Yaskawa INFORM job: A_ROOF_UPPER_0614_2_PAINT_51.JBI

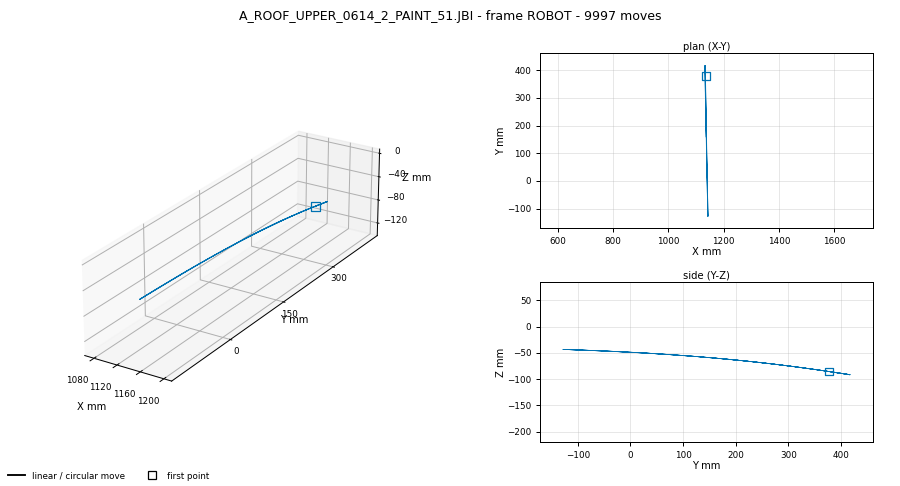
[picture p0: tool path of A_ROOF_UPPER_0614_2_PAINT_51.JBI in frame ROBOT, 9997 of 9997 moves have a stored position in this frame; points joined in program order, loops and branches not executed]
/JOB
//NAME A_ROOF_UPPER_0614_2_PAINT51
//POS
///NPOS 9997,0,0,0,0,0
///TOOL 1
///USER 0
///POSTYPE ROBOT
///RECTAN
///RCONF 1,0,0,0,0,0,0,0,0,0,0,0,0,0,0,0,0,0,0,0,0,0,0,0
C00000=1135.150,378.106,-85.384,-176.923,11.211,149.474
C00001=1135.147,378.354,-85.422,-176.921,11.213,149.474
C00002=1135.142,378.601,-85.459,-176.917,11.216,149.474
C00003=1135.138,378.848,-85.496,-176.915,11.218,149.474
C00004=1135.135,379.096,-85.533,-176.913,11.220,149.474
C00005=1135.131,379.342,-85.571,-176.910,11.222,149.474
C00006=1135.127,379.590,-85.608,-176.907,11.224,149.474
C00007=1135.124,379.837,-85.645,-176.904,11.227,149.474
C00008=1135.120,380.084,-85.682,-176.902,11.229,149.474
C00009=1135.116,380.331,-85.719,-176.899,11.231,149.473
C00010=1135.112,380.578,-85.756,-176.896,11.234,149.473
C00011=1135.108,380.826,-85.794,-176.894,11.236,149.473
C00012=1135.104,381.073,-85.831,-176.891,11.239,149.473
C00013=1135.101,381.320,-85.869,-176.889,11.241,149.473
C00014=1135.097,381.567,-85.906,-176.887,11.243,149.473
C00015=1135.093,381.814,-85.943,-176.883,11.245,149.473
C00016=1135.090,382.062,-85.981,-176.881,11.247,149.473
C00017=1135.086,382.309,-86.017,-176.879,11.249,149.473
C00018=1135.082,382.556,-86.055,-176.876,11.252,149.473
C00019=1135.078,382.803,-86.092,-176.874,11.254,149.473
C00020=1135.075,383.050,-86.130,-176.871,11.256,149.473
C00021=1135.070,383.297,-86.167,-176.869,11.259,149.473
C00022=1135.067,383.545,-86.205,-176.867,11.260,149.473
C00023=1135.063,383.792,-86.241,-176.866,11.262,149.473
C00024=1135.060,384.039,-86.279,-176.865,11.264,149.473
C00025=1135.056,384.286,-86.317,-176.865,11.265,149.473
C00026=1135.052,384.533,-86.354,-176.863,11.266,149.473
C00027=1135.049,384.780,-86.392,-176.862,11.268,149.473
C00028=1135.045,385.027,-86.429,-176.861,11.270,149.474
C00029=1135.042,385.274,-86.467,-176.861,11.271,149.474
C00030=1135.037,385.522,-86.504,-176.860,11.272,149.474
C00031=1135.033,385.769,-86.542,-176.859,11.274,149.474
C00032=1135.030,386.016,-86.580,-176.858,11.276,149.474
C00033=1135.026,386.263,-86.616,-176.857,11.277,149.475
C00034=1135.023,386.510,-86.654,-176.856,11.279,149.475
C00035=1135.018,386.757,-86.691,-176.855,11.280,149.475
C00036=1135.015,387.005,-86.729,-176.854,11.282,149.475
C00037=1135.011,387.252,-86.766,-176.854,11.283,149.476
C00038=1135.007,387.498,-86.804,-176.853,11.285,149.476
C00039=1135.004,387.746,-86.842,-176.853,11.287,149.476
C00040=1134.999,387.993,-86.879,-176.852,11.289,149.476
C00041=1134.996,388.241,-86.917,-176.851,11.290,149.477
C00042=1134.992,388.487,-86.954,-176.851,11.292,149.477
C00043=1134.989,388.700,-86.986,-176.850,11.294,149.477
C00044=1134.986,388.913,-87.019,-176.850,11.295,149.477
C00045=1134.983,389.126,-87.051,-176.849,11.297,149.478
C00046=1134.980,389.339,-87.084,-176.848,11.298,149.478
C00047=1134.976,389.551,-87.116,-176.848,11.300,149.478
C00048=1134.973,389.764,-87.148,-176.847,11.301,149.478
C00049=1134.970,389.977,-87.180,-176.846,11.303,149.479
C00050=1134.967,390.189,-87.213,-176.847,11.305,149.479
C00051=1134.963,390.437,-87.250,-176.846,11.306,149.479
C00052=1134.960,390.684,-87.288,-176.845,11.309,149.480
C00053=1134.956,390.931,-87.326,-176.845,11.310,149.480
C00054=1134.952,391.178,-87.363,-176.845,11.312,149.481
C00055=1134.948,391.426,-87.401,-176.844,11.314,149.481
C00056=1134.945,391.672,-87.439,-176.843,11.316,149.481
C00057=1134.941,391.919,-87.476,-176.844,11.318,149.482
C00058=1134.937,392.167,-87.513,-176.843,11.320,149.482
C00059=1134.933,392.414,-87.552,-176.843,11.322,149.483
C00060=1134.930,392.661,-87.590,-176.842,11.324,149.483
C00061=1134.926,392.908,-87.626,-176.842,11.326,149.483
C00062=1134.922,393.155,-87.664,-176.842,11.328,149.484
C00063=1134.919,393.402,-87.702,-176.841,11.330,149.484
C00064=1134.915,393.650,-87.739,-176.841,11.332,149.485
C00065=1134.911,393.897,-87.777,-176.841,11.334,149.485
C00066=1134.907,394.144,-87.815,-176.841,11.336,149.486
C00067=1134.904,394.391,-87.853,-176.841,11.339,149.486
C00068=1134.900,394.638,-87.890,-176.840,11.341,149.487
C00069=1134.896,394.885,-87.928,-176.840,11.342,149.487
C00070=1134.892,395.133,-87.966,-176.840,11.345,149.488
C00071=1134.889,395.379,-88.004,-176.840,11.347,149.488
C00072=1134.884,395.626,-88.041,-176.840,11.350,149.489
C00073=1134.881,395.874,-88.079,-176.840,11.352,149.490
C00074=1134.878,396.120,-88.116,-176.840,11.354,149.490
C00075=1134.874,396.368,-88.155,-176.840,11.356,149.491
C00076=1134.870,396.614,-88.192,-176.840,11.359,149.491
C00077=1134.866,396.862,-88.229,-176.840,11.361,149.492
C00078=1134.863,397.109,-88.267,-176.839,11.364,149.493
C00079=1134.859,397.356,-88.306,-176.840,11.366,149.493
C00080=1134.855,397.603,-88.343,-176.840,11.368,149.494
C00081=1134.852,397.850,-88.381,-176.840,11.371,149.495
C00082=1134.848,398.097,-88.418,-176.840,11.373,149.495
C00083=1134.844,398.345,-88.456,-176.840,11.376,149.496
C00084=1134.840,398.592,-88.494,-176.840,11.378,149.496
C00085=1134.837,398.839,-88.532,-176.841,11.381,149.497
C00086=1134.833,399.085,-88.570,-176.841,11.383,149.498
C00087=1134.829,399.334,-88.607,-176.841,11.386,149.499
C00088=1134.825,399.580,-88.645,-176.841,11.389,149.499
C00089=1134.822,399.827,-88.683,-176.842,11.391,149.500
C00090=1134.818,400.074,-88.720,-176.842,11.393,149.501
C00091=1134.814,400.322,-88.759,-176.842,11.396,149.502
C00092=1134.810,400.568,-88.797,-176.842,11.399,149.502
C00093=1134.807,400.815,-88.835,-176.843,11.402,149.503
C00094=1134.803,401.063,-88.871,-176.843,11.405,149.504
C00095=1134.799,401.310,-88.910,-176.843,11.407,149.505
C00096=1134.795,401.557,-88.947,-176.844,11.409,149.506
C00097=1134.792,401.804,-88.985,-176.845,11.413,149.507
C00098=1134.788,402.051,-89.023,-176.845,11.416,149.507
C00099=1134.785,402.264,-89.056,-176.845,11.418,149.508
C00100=1134.782,402.476,-89.089,-176.846,11.420,149.509
C00101=1134.779,402.690,-89.121,-176.846,11.423,149.510
C00102=1134.775,402.902,-89.153,-176.846,11.426,149.510
C00103=1134.772,403.114,-89.186,-176.847,11.428,149.511
C00104=1134.769,403.327,-89.219,-176.847,11.431,149.512
C00105=1134.765,403.540,-89.251,-176.848,11.433,149.513
C00106=1134.762,403.753,-89.284,-176.849,11.436,149.514
C00107=1134.759,403.999,-89.322,-176.849,11.439,149.515
C00108=1134.755,404.247,-89.359,-176.850,11.442,149.515
C00109=1134.751,404.494,-89.397,-176.850,11.445,149.516
C00110=1134.747,404.741,-89.435,-176.851,11.448,149.517
C00111=1134.744,404.988,-89.473,-176.852,11.451,149.518
C00112=1134.740,405.235,-89.511,-176.852,11.455,149.519
C00113=1134.736,405.482,-89.549,-176.854,11.457,149.520
C00114=1134.733,405.729,-89.587,-176.854,11.460,149.521
C00115=1134.730,405.977,-89.625,-176.855,11.464,149.522
C00116=1134.725,406.224,-89.663,-176.856,11.467,149.523
C00117=1134.722,406.471,-89.701,-176.857,11.470,149.525
C00118=1134.718,406.717,-89.739,-176.858,11.473,149.526
C00119=1134.715,406.965,-89.777,-176.859,11.477,149.527
C00120=1134.710,407.212,-89.815,-176.859,11.480,149.528
C00121=1134.707,407.459,-89.852,-176.861,11.484,149.529
C00122=1134.703,407.706,-89.889,-176.861,11.487,149.530
C00123=1134.699,407.954,-89.928,-176.862,11.491,149.531
C00124=1134.695,408.200,-89.966,-176.863,11.494,149.532
C00125=1134.692,408.447,-90.004,-176.865,11.498,149.534
C00126=1134.688,408.694,-90.042,-176.866,11.501,149.535
C00127=1134.684,408.942,-90.080,-176.867,11.505,149.536
C00128=1134.681,409.189,-90.118,-176.868,11.508,149.537
C00129=1134.677,409.436,-90.156,-176.869,11.512,149.538
C00130=1134.674,409.683,-90.194,-176.870,11.515,149.540
C00131=1134.670,409.930,-90.231,-176.871,11.519,149.541
C00132=1134.666,410.177,-90.270,-176.873,11.523,149.542
C00133=1134.662,410.424,-90.307,-176.874,11.526,149.543
C00134=1134.659,410.671,-90.345,-176.875,11.530,149.545
C00135=1134.654,410.918,-90.383,-176.876,11.534,149.546
C00136=1134.651,411.165,-90.421,-176.877,11.538,149.547
C00137=1134.648,411.412,-90.459,-176.879,11.542,149.549
C00138=1134.643,411.659,-90.498,-176.880,11.546,149.550
C00139=1134.640,411.907,-90.535,-176.881,11.550,149.551
C00140=1134.636,412.153,-90.573,-176.883,11.554,149.553
C00141=1134.633,412.401,-90.612,-176.884,11.558,149.554
C00142=1134.629,412.647,-90.649,-176.886,11.562,149.556
C00143=1134.626,412.895,-90.687,-176.887,11.566,149.557
C00144=1134.621,413.141,-90.725,-176.889,11.569,149.558
C00145=1134.618,413.389,-90.763,-176.890,11.573,149.560
C00146=1134.615,413.636,-90.801,-176.892,11.578,149.561
C00147=1134.610,413.883,-90.839,-176.893,11.582,149.563
C00148=1134.607,414.130,-90.877,-176.895,11.586,149.564
C00149=1134.603,414.377,-90.915,-176.896,11.590,149.566
C00150=1134.600,414.624,-90.953,-176.898,11.595,149.567
C00151=1134.598,414.871,-90.991,-176.900,11.599,149.569
C00152=1134.597,415.119,-91.029,-176.901,11.604,149.571
C00153=1134.596,415.365,-91.067,-176.903,11.608,149.572
C00154=1134.595,415.613,-91.104,-176.905,11.612,149.574
C00155=1134.595,415.825,-91.136,-176.907,11.616,149.575
C00156=1134.596,416.038,-91.169,-176.908,11.620,149.576
C00157=1134.597,416.250,-91.201,-176.910,11.623,149.578
C00158=1134.599,416.463,-91.233,-176.912,11.627,149.579
C00159=1134.601,416.676,-91.265,-176.913,11.631,149.581
C00160=1134.603,416.888,-91.296,-176.915,11.635,149.582
C00161=1134.606,417.101,-91.328,-176.917,11.639,149.584
C00162=1134.609,417.314,-91.359,-176.919,11.642,149.585
C00163=1134.191,417.313,-91.423,-176.911,11.647,149.584
C00164=1134.187,417.101,-91.391,-176.909,11.643,149.583
C00165=1134.184,416.888,-91.359,-176.907,11.639,149.581
C00166=1134.181,416.675,-91.327,-176.906,11.635,149.580
C00167=1134.179,416.462,-91.295,-176.905,11.631,149.579
C00168=1134.178,416.250,-91.263,-176.903,11.628,149.577
C00169=1134.176,416.037,-91.231,-176.901,11.623,149.576
C00170=1134.176,415.825,-91.199,-176.900,11.620,149.574
C00171=1134.176,415.613,-91.167,-176.898,11.616,149.573
C00172=1134.176,415.365,-91.128,-176.896,11.611,149.571
C00173=1134.177,415.118,-91.091,-176.895,11.607,149.570
C00174=1134.179,414.871,-91.053,-176.893,11.603,149.568
C00175=1134.181,414.624,-91.016,-176.891,11.599,149.567
C00176=1134.184,414.377,-90.978,-176.889,11.595,149.565
C00177=1134.187,414.129,-90.940,-176.889,11.590,149.564
C00178=1134.191,413.883,-90.902,-176.887,11.586,149.562
C00179=1134.194,413.636,-90.864,-176.885,11.582,149.561
C00180=1134.198,413.388,-90.826,-176.883,11.578,149.559
C00181=1134.202,413.141,-90.788,-176.883,11.573,149.558
C00182=1134.206,412.894,-90.749,-176.881,11.569,149.556
C00183=1134.209,412.648,-90.711,-176.880,11.566,149.555
C00184=1134.213,412.401,-90.673,-176.878,11.561,149.554
C00185=1134.217,412.154,-90.635,-176.876,11.557,149.552
C00186=1134.220,411.907,-90.597,-176.875,11.554,149.551
C00187=1134.224,411.659,-90.559,-176.874,11.549,149.550
C00188=1134.228,411.412,-90.521,-176.873,11.545,149.548
C00189=1134.231,411.165,-90.483,-176.871,11.541,149.547
C00190=1134.235,410.919,-90.446,-176.870,11.538,149.546
C00191=1134.239,410.671,-90.407,-176.869,11.534,149.544
C00192=1134.243,410.424,-90.369,-176.868,11.531,149.543
C00193=1134.247,410.177,-90.331,-176.866,11.527,149.542
C00194=1134.250,409.930,-90.293,-176.866,11.522,149.540
C00195=1134.254,409.683,-90.255,-176.865,11.519,149.539
C00196=1134.258,409.435,-90.217,-176.863,11.515,149.538
C00197=1134.261,409.189,-90.179,-176.862,11.511,149.537
C00198=1134.265,408.942,-90.141,-176.861,11.508,149.535
C00199=1134.269,408.695,-90.103,-176.860,11.504,149.534
C00200=1134.272,408.447,-90.065,-176.859,11.501,149.533
C00201=1134.276,408.201,-90.028,-176.858,11.497,149.532
C00202=1134.280,407.953,-89.989,-176.857,11.494,149.531
C00203=1134.283,407.706,-89.951,-176.856,11.490,149.530
C00204=1134.287,407.459,-89.914,-176.855,11.487,149.529
C00205=1134.290,407.212,-89.876,-176.854,11.484,149.527
C00206=1134.295,406.965,-89.838,-176.853,11.480,149.526
C00207=1134.298,406.717,-89.800,-176.852,11.477,149.525
C00208=1134.302,406.471,-89.763,-176.852,11.474,149.524
C00209=1134.306,406.223,-89.724,-176.850,11.470,149.523
C00210=1134.310,405.977,-89.687,-176.850,11.467,149.522
C00211=1134.313,405.729,-89.649,-176.849,11.464,149.521
C00212=1134.317,405.482,-89.610,-176.848,11.460,149.520
C00213=1134.321,405.235,-89.573,-176.848,11.457,149.519
C00214=1134.324,404.988,-89.535,-176.847,11.454,149.518
C00215=1134.328,404.741,-89.496,-176.846,11.451,149.517
C00216=1134.332,404.494,-89.458,-176.846,11.448,149.516
C00217=1134.335,404.247,-89.421,-176.845,11.445,149.515
C00218=1134.338,404.000,-89.383,-176.845,11.441,149.514
C00219=1134.343,403.753,-89.345,-176.844,11.438,149.513
C00220=1134.346,403.540,-89.312,-176.844,11.436,149.512
C00221=1134.350,403.327,-89.280,-176.843,11.434,149.512
C00222=1134.353,403.115,-89.247,-176.843,11.431,149.511
C00223=1134.355,402.902,-89.215,-176.842,11.428,149.510
C00224=1134.359,402.690,-89.182,-176.841,11.426,149.509
C00225=1134.362,402.477,-89.149,-176.841,11.423,149.509
C00226=1134.365,402.264,-89.117,-176.841,11.420,149.508
C00227=1134.368,402.051,-89.084,-176.841,11.419,149.507
C00228=1134.372,401.805,-89.046,-176.840,11.415,149.506
C00229=1134.376,401.556,-89.009,-176.840,11.412,149.505
C00230=1134.380,401.310,-88.971,-176.839,11.410,149.504
C00231=1134.383,401.063,-88.933,-176.839,11.407,149.504
C00232=1134.387,400.816,-88.895,-176.839,11.404,149.503
C00233=1134.391,400.568,-88.857,-176.839,11.401,149.502
C00234=1134.394,400.322,-88.819,-176.838,11.398,149.501
C00235=1134.398,400.075,-88.781,-176.838,11.395,149.500
C00236=1134.401,399.828,-88.744,-176.838,11.393,149.500
C00237=1134.406,399.580,-88.706,-176.837,11.391,149.499
C00238=1134.409,399.333,-88.668,-176.837,11.388,149.498
C00239=1134.413,399.086,-88.630,-176.837,11.385,149.498
C00240=1134.416,398.839,-88.593,-176.837,11.383,149.497
C00241=1134.420,398.592,-88.554,-176.837,11.380,149.496
C00242=1134.424,398.345,-88.517,-176.837,11.378,149.496
C00243=1134.428,398.097,-88.480,-176.837,11.375,149.495
C00244=1134.431,397.851,-88.442,-176.837,11.372,149.494
C00245=1134.435,397.603,-88.403,-176.836,11.370,149.494
C00246=1134.439,397.357,-88.366,-176.836,11.368,149.493
C00247=1134.442,397.109,-88.328,-176.836,11.365,149.492
C00248=1134.446,396.862,-88.291,-176.836,11.363,149.492
C00249=1134.450,396.615,-88.253,-176.837,11.360,149.491
C00250=1134.454,396.368,-88.215,-176.837,11.358,149.490
C00251=1134.457,396.121,-88.177,-176.836,11.356,149.490
C00252=1134.461,395.874,-88.139,-176.837,11.354,149.489
C00253=1134.465,395.626,-88.102,-176.837,11.351,149.489
C00254=1134.469,395.379,-88.064,-176.837,11.349,149.488
C00255=1134.472,395.132,-88.026,-176.837,11.347,149.488
C00256=1134.476,394.886,-87.989,-176.838,11.344,149.487
C00257=1134.480,394.639,-87.951,-176.837,11.343,149.487
C00258=1134.484,394.391,-87.913,-176.838,11.340,149.486
C00259=1134.488,394.144,-87.876,-176.838,11.338,149.485
C00260=1134.491,393.897,-87.838,-176.838,11.336,149.485
C00261=1134.495,393.650,-87.800,-176.839,11.333,149.485
C00262=1134.498,393.402,-87.763,-176.839,11.332,149.484
C00263=1134.503,393.156,-87.725,-176.839,11.330,149.484
C00264=1134.506,392.908,-87.687,-176.840,11.327,149.483
C00265=1134.510,392.662,-87.649,-176.840,11.325,149.483
C00266=1134.513,392.414,-87.612,-176.841,11.323,149.482
C00267=1134.517,392.167,-87.574,-176.840,11.322,149.482
C00268=1134.521,391.920,-87.536,-176.841,11.319,149.481
C00269=1134.525,391.673,-87.499,-176.841,11.317,149.481
C00270=1134.528,391.425,-87.461,-176.842,11.315,149.481
C00271=1134.532,391.179,-87.423,-176.843,11.313,149.480
C00272=1134.536,390.932,-87.386,-176.842,11.312,149.480
C00273=1134.539,390.684,-87.349,-176.843,11.310,149.480
C00274=1134.543,390.438,-87.311,-176.844,11.307,149.479
C00275=1134.547,390.190,-87.273,-176.845,11.306,149.479
C00276=1134.550,389.977,-87.241,-176.845,11.304,149.479
C00277=1134.553,389.764,-87.208,-176.846,11.302,149.478
C00278=1134.557,389.552,-87.176,-176.846,11.301,149.478
C00279=1134.560,389.339,-87.144,-176.846,11.299,149.478
C00280=1134.563,389.126,-87.111,-176.847,11.298,149.477
C00281=1134.566,388.913,-87.080,-176.847,11.296,149.477
C00282=1134.570,388.701,-87.047,-176.848,11.294,149.477
C00283=1134.573,388.488,-87.014,-176.849,11.293,149.477
C00284=1134.577,388.241,-86.977,-176.849,11.291,149.476
C00285=1134.580,387.993,-86.939,-176.850,11.289,149.476
C00286=1134.584,387.747,-86.902,-176.851,11.288,149.476
C00287=1134.587,387.499,-86.865,-176.852,11.287,149.476
C00288=1134.592,387.252,-86.826,-176.853,11.285,149.475
C00289=1134.596,387.005,-86.790,-176.853,11.283,149.475
C00290=1134.599,386.758,-86.752,-176.854,11.281,149.475
C00291=1134.603,386.511,-86.714,-176.855,11.280,149.475
C00292=1134.606,386.263,-86.677,-176.856,11.278,149.475
C00293=1134.610,386.017,-86.639,-176.857,11.276,149.474
C00294=1134.614,385.769,-86.602,-176.858,11.274,149.474
C00295=1134.617,385.522,-86.564,-176.858,11.274,149.474
C00296=1134.621,385.276,-86.527,-176.859,11.272,149.474
C00297=1134.625,385.028,-86.490,-176.860,11.270,149.474
C00298=1134.628,384.781,-86.452,-176.861,11.269,149.474
C00299=1134.633,384.533,-86.414,-176.862,11.267,149.473
C00300=1134.636,384.286,-86.377,-176.863,11.266,149.473
C00301=1134.641,384.039,-86.340,-176.864,11.264,149.473
C00302=1134.644,383.792,-86.302,-176.865,11.262,149.473
C00303=1134.648,383.545,-86.265,-176.866,11.261,149.473
C00304=1134.651,383.297,-86.227,-176.868,11.259,149.473
C00305=1134.655,383.051,-86.189,-176.870,11.256,149.473
C00306=1134.659,382.804,-86.153,-176.873,11.254,149.473
C00307=1134.662,382.556,-86.115,-176.875,11.252,149.473
C00308=1134.666,382.309,-86.078,-176.878,11.250,149.473
C00309=1134.670,382.062,-86.041,-176.881,11.248,149.473
C00310=1134.673,381.815,-86.003,-176.883,11.246,149.473
C00311=1134.678,381.568,-85.966,-176.886,11.243,149.473
C00312=1134.681,381.320,-85.928,-176.888,11.241,149.473
C00313=1134.685,381.073,-85.891,-176.890,11.239,149.473
C00314=1134.689,380.827,-85.854,-176.893,11.236,149.473
C00315=1134.692,380.579,-85.817,-176.895,11.234,149.473
C00316=1134.696,380.331,-85.780,-176.899,11.232,149.474
C00317=1134.700,380.085,-85.742,-176.901,11.230,149.474
C00318=1134.704,379.837,-85.705,-176.903,11.228,149.474
C00319=1134.708,379.590,-85.668,-176.906,11.225,149.474
C00320=1134.711,379.343,-85.630,-176.909,11.223,149.474
C00321=1134.715,379.095,-85.593,-176.912,11.220,149.474
C00322=1134.719,378.848,-85.556,-176.914,11.218,149.474
C00323=1134.723,378.602,-85.519,-176.917,11.216,149.474
C00324=1134.727,378.354,-85.482,-176.920,11.214,149.474
C00325=1134.730,378.107,-85.445,-176.922,11.212,149.474
C00326=1134.733,377.860,-85.408,-176.925,11.209,149.474
C00327=1134.738,377.613,-85.371,-176.927,11.207,149.475
C00328=1134.741,377.365,-85.334,-176.931,11.205,149.475
C00329=1134.745,377.118,-85.297,-176.933,11.203,149.475
C00330=1134.749,376.871,-85.260,-176.936,11.200,149.475
C00331=1134.753,376.624,-85.222,-176.939,11.198,149.475
C00332=1134.755,376.411,-85.191,-176.941,11.197,149.475
C00333=1134.759,376.198,-85.159,-176.944,11.195,149.475
C00334=1134.763,375.985,-85.127,-176.946,11.192,149.475
C00335=1134.766,375.772,-85.096,-176.948,11.191,149.476
C00336=1134.769,375.559,-85.063,-176.951,11.189,149.476
C00337=1134.772,375.347,-85.031,-176.953,11.187,149.476
C00338=1134.776,375.134,-85.000,-176.956,11.185,149.476
C00339=1134.779,374.921,-84.968,-176.958,11.183,149.476
C00340=1134.782,374.673,-84.931,-176.961,11.181,149.476
C00341=1134.786,374.426,-84.894,-176.964,11.178,149.476
C00342=1134.790,374.179,-84.857,-176.967,11.176,149.477
C00343=1134.794,373.932,-84.821,-176.970,11.174,149.477
C00344=1134.798,373.685,-84.784,-176.972,11.172,149.477
C00345=1134.801,373.437,-84.747,-176.976,11.169,149.477
C00346=1134.806,373.190,-84.710,-176.978,11.167,149.477
C00347=1134.809,372.943,-84.674,-176.982,11.165,149.477
C00348=1134.813,372.695,-84.637,-176.985,11.162,149.477
C00349=1134.817,372.448,-84.600,-176.987,11.160,149.478
C00350=1134.821,372.200,-84.563,-176.991,11.158,149.478
C00351=1134.824,371.953,-84.527,-176.993,11.156,149.478
C00352=1134.828,371.706,-84.490,-176.997,11.154,149.478
C00353=1134.832,371.459,-84.453,-176.999,11.151,149.478
C00354=1134.835,371.212,-84.417,-177.002,11.149,149.479
C00355=1134.840,370.965,-84.380,-177.005,11.147,149.479
C00356=1134.843,370.717,-84.343,-177.009,11.144,149.479
C00357=1134.846,370.470,-84.306,-177.011,11.143,149.479
C00358=1134.850,370.223,-84.270,-177.015,11.140,149.480
C00359=1134.855,369.975,-84.233,-177.018,11.138,149.480
C00360=1134.858,369.728,-84.197,-177.021,11.136,149.480
C00361=1134.862,369.481,-84.160,-177.024,11.133,149.480
C00362=1134.866,369.234,-84.123,-177.027,11.131,149.480
C00363=1134.869,368.986,-84.087,-177.030,11.128,149.480
C00364=1134.874,368.739,-84.051,-177.033,11.126,149.481
C00365=1134.877,368.492,-84.014,-177.036,11.124,149.481
C00366=1134.881,368.245,-83.978,-177.039,11.122,149.481
C00367=1134.885,367.997,-83.941,-177.043,11.119,149.481
C00368=1134.889,367.750,-83.905,-177.045,11.117,149.482
C00369=1134.893,367.503,-83.868,-177.049,11.115,149.482
C00370=1134.896,367.256,-83.832,-177.052,11.112,149.482
C00371=1134.901,367.008,-83.796,-177.055,11.110,149.482
C00372=1134.904,366.761,-83.760,-177.058,11.109,149.483
C00373=1134.908,366.514,-83.723,-177.062,11.106,149.483
C00374=1134.912,366.265,-83.686,-177.065,11.104,149.483
C00375=1134.915,366.018,-83.650,-177.068,11.101,149.483
C00376=1134.920,365.771,-83.614,-177.072,11.099,149.483
C00377=1134.923,365.524,-83.578,-177.075,11.096,149.484
C00378=1134.927,365.277,-83.541,-177.078,11.095,149.484
C00379=1134.931,365.029,-83.505,-177.081,11.092,149.484
C00380=1134.934,364.782,-83.469,-177.084,11.090,149.484
C00381=1134.939,364.534,-83.433,-177.088,11.087,149.485
C00382=1134.942,364.288,-83.396,-177.091,11.085,149.485
C00383=1134.946,364.040,-83.360,-177.095,11.083,149.485
C00384=1134.950,363.793,-83.324,-177.098,11.080,149.485
C00385=1134.954,363.545,-83.288,-177.101,11.078,149.486
C00386=1134.957,363.298,-83.252,-177.104,11.075,149.486
C00387=1134.961,363.051,-83.216,-177.107,11.073,149.486
C00388=1134.965,362.838,-83.184,-177.110,11.071,149.486
C00389=1134.968,362.624,-83.154,-177.113,11.069,149.487
C00390=1134.971,362.412,-83.122,-177.116,11.067,149.487
C00391=1134.975,362.198,-83.092,-177.119,11.065,149.487
C00392=1134.978,361.986,-83.061,-177.122,11.063,149.487
C00393=1134.981,361.773,-83.030,-177.125,11.061,149.488
C00394=1134.985,361.560,-82.998,-177.128,11.059,149.488
C00395=1134.988,361.346,-82.968,-177.131,11.057,149.488
C00396=1134.991,361.099,-82.931,-177.134,11.054,149.488
C00397=1134.995,360.852,-82.896,-177.138,11.052,149.488
C00398=1135.000,360.604,-82.860,-177.141,11.049,149.489
C00399=1135.003,360.357,-82.824,-177.145,11.047,149.489
C00400=1135.007,360.110,-82.788,-177.148,11.045,149.489
C00401=1135.010,359.862,-82.752,-177.151,11.042,149.489
C00402=1135.015,359.614,-82.716,-177.155,11.040,149.490
C00403=1135.018,359.367,-82.681,-177.158,11.038,149.490
C00404=1135.022,359.120,-82.644,-177.162,11.035,149.490
C00405=1135.026,358.872,-82.608,-177.165,11.033,149.491
C00406=1135.030,358.625,-82.573,-177.169,11.030,149.491
C00407=1135.034,358.378,-82.537,-177.173,11.027,149.491
C00408=1135.038,358.130,-82.502,-177.176,11.025,149.491
C00409=1135.041,357.883,-82.466,-177.179,11.022,149.492
C00410=1135.045,357.636,-82.429,-177.183,11.020,149.492
C00411=1135.049,357.388,-82.394,-177.186,11.018,149.492
C00412=1135.053,357.141,-82.358,-177.190,11.015,149.492
C00413=1135.056,356.893,-82.323,-177.194,11.012,149.493
C00414=1135.060,356.646,-82.287,-177.197,11.010,149.493
C00415=1135.065,356.399,-82.252,-177.200,11.008,149.493
C00416=1135.069,356.151,-82.216,-177.204,11.005,149.494
C00417=1135.072,355.904,-82.180,-177.208,11.002,149.494
C00418=1135.076,355.656,-82.145,-177.211,11.000,149.494
C00419=1135.080,355.409,-82.109,-177.215,10.998,149.494
C00420=1135.083,355.161,-82.074,-177.218,10.995,149.495
C00421=1135.088,354.914,-82.039,-177.222,10.992,149.495
C00422=1135.091,354.667,-82.003,-177.226,10.989,149.495
C00423=1135.095,354.419,-81.968,-177.229,10.987,149.495
C00424=1135.100,354.171,-81.932,-177.233,10.984,149.496
C00425=1135.104,353.924,-81.897,-177.237,10.982,149.496
C00426=1135.108,353.677,-81.861,-177.240,10.979,149.496
C00427=1135.111,353.429,-81.826,-177.244,10.976,149.497
C00428=1135.115,353.182,-81.790,-177.248,10.974,149.497
C00429=1135.119,352.934,-81.755,-177.251,10.972,149.497
C00430=1135.123,352.687,-81.720,-177.255,10.968,149.497
C00431=1135.127,352.439,-81.685,-177.258,10.966,149.498
C00432=1135.130,352.192,-81.649,-177.263,10.963,149.498
C00433=1135.134,351.944,-81.614,-177.266,10.961,149.498
C00434=1135.139,351.697,-81.579,-177.269,10.958,149.498
C00435=1135.142,351.449,-81.544,-177.274,10.955,149.499
C00436=1135.146,351.202,-81.508,-177.277,10.953,149.499
C00437=1135.151,350.954,-81.474,-177.281,10.949,149.499
C00438=1135.154,350.707,-81.438,-177.285,10.947,149.500
C00439=1135.158,350.459,-81.402,-177.289,10.944,149.500
C00440=1135.162,350.212,-81.369,-177.292,10.942,149.500
C00441=1135.165,349.965,-81.333,-177.296,10.939,149.500
C00442=1135.169,349.717,-81.297,-177.300,10.936,149.501
C00443=1135.174,349.470,-81.263,-177.304,10.933,149.501
C00444=1135.177,349.257,-81.232,-177.306,10.931,149.501
C00445=1135.180,349.043,-81.202,-177.310,10.929,149.501
C00446=1135.184,348.829,-81.172,-177.312,10.927,149.501
C00447=1135.187,348.616,-81.142,-177.315,10.924,149.502
C00448=1135.191,348.404,-81.112,-177.317,10.922,149.502
C00449=1135.194,348.191,-81.081,-177.320,10.921,149.502
C00450=1135.197,347.977,-81.052,-177.323,10.918,149.502
C00451=1135.200,347.764,-81.022,-177.326,10.916,149.502
C00452=1135.204,347.517,-80.986,-177.329,10.914,149.502
C00453=1135.208,347.269,-80.952,-177.332,10.911,149.503
C00454=1135.212,347.021,-80.917,-177.336,10.909,149.503
C00455=1135.216,346.774,-80.882,-177.339,10.906,149.503
C00456=1135.220,346.526,-80.847,-177.342,10.904,149.503
C00457=1135.224,346.279,-80.812,-177.346,10.902,149.504
C00458=1135.228,346.031,-80.777,-177.349,10.899,149.504
C00459=1135.232,345.783,-80.742,-177.352,10.896,149.504
C00460=1135.236,345.536,-80.708,-177.355,10.894,149.504
C00461=1135.240,345.288,-80.673,-177.359,10.891,149.504
C00462=1135.244,345.041,-80.639,-177.362,10.889,149.505
C00463=1135.248,344.793,-80.603,-177.365,10.886,149.505
C00464=1135.252,344.546,-80.569,-177.368,10.884,149.505
C00465=1135.256,344.298,-80.534,-177.372,10.882,149.505
C00466=1135.260,344.050,-80.499,-177.375,10.879,149.505
C00467=1135.263,343.804,-80.465,-177.378,10.876,149.506
C00468=1135.267,343.555,-80.430,-177.381,10.874,149.506
C00469=1135.272,343.308,-80.396,-177.385,10.871,149.506
C00470=1135.275,343.060,-80.361,-177.388,10.869,149.506
C00471=1135.279,342.813,-80.327,-177.391,10.866,149.507
C00472=1135.283,342.565,-80.291,-177.395,10.864,149.507
C00473=1135.287,342.318,-80.257,-177.397,10.861,149.507
C00474=1135.291,342.070,-80.223,-177.401,10.859,149.507
C00475=1135.296,341.823,-80.188,-177.404,10.856,149.507
C00476=1135.299,341.575,-80.154,-177.407,10.854,149.508
C00477=1135.303,341.327,-80.119,-177.411,10.851,149.508
C00478=1135.307,341.079,-80.085,-177.414,10.849,149.508
C00479=1135.311,340.832,-80.051,-177.417,10.846,149.508
C00480=1135.316,340.585,-80.016,-177.420,10.844,149.508
C00481=1135.319,340.337,-79.982,-177.424,10.841,149.508
C00482=1135.323,340.090,-79.948,-177.427,10.839,149.509
C00483=1135.327,339.842,-79.913,-177.430,10.836,149.509
C00484=1135.331,339.594,-79.879,-177.434,10.834,149.509
C00485=1135.335,339.346,-79.844,-177.436,10.831,149.509
C00486=1135.339,339.099,-79.810,-177.440,10.829,149.509
C00487=1135.343,338.851,-79.775,-177.443,10.826,149.510
C00488=1135.347,338.604,-79.741,-177.446,10.824,149.510
C00489=1135.351,338.356,-79.707,-177.450,10.821,149.510
C00490=1135.355,338.109,-79.673,-177.453,10.819,149.510
C00491=1135.359,337.861,-79.638,-177.456,10.816,149.510
C00492=1135.362,337.613,-79.604,-177.459,10.814,149.511
C00493=1135.367,337.366,-79.570,-177.463,10.811,149.511
C00494=1135.371,337.119,-79.536,-177.466,10.809,149.511
C00495=1135.374,336.870,-79.502,-177.469,10.806,149.511
C00496=1135.379,336.623,-79.468,-177.472,10.803,149.512
C00497=1135.382,336.375,-79.433,-177.476,10.801,149.512
C00498=1135.387,336.128,-79.399,-177.479,10.799,149.512
C00499=1135.391,335.881,-79.365,-177.482,10.797,149.512
C00500=1135.394,335.667,-79.336,-177.484,10.794,149.512
C00501=1135.397,335.453,-79.306,-177.487,10.792,149.513
C00502=1135.401,335.240,-79.277,-177.490,10.790,149.513
C00503=1135.404,335.027,-79.248,-177.493,10.788,149.513
C00504=1135.408,334.814,-79.218,-177.496,10.785,149.513
C00505=1135.411,334.600,-79.189,-177.498,10.784,149.513
C00506=1135.414,334.387,-79.160,-177.501,10.782,149.513
C00507=1135.418,334.173,-79.130,-177.504,10.779,149.514
C00508=1135.422,333.925,-79.097,-177.507,10.777,149.514
C00509=1135.425,333.678,-79.063,-177.510,10.774,149.514
C00510=1135.430,333.430,-79.029,-177.514,10.771,149.514
C00511=1135.434,333.182,-78.995,-177.517,10.769,149.514
C00512=1135.438,332.935,-78.962,-177.520,10.767,149.515
C00513=1135.441,332.688,-78.927,-177.523,10.764,149.515
C00514=1135.446,332.439,-78.894,-177.526,10.761,149.515
C00515=1135.450,332.192,-78.860,-177.530,10.759,149.515
C00516=1135.453,331.944,-78.826,-177.533,10.756,149.515
C00517=1135.458,331.697,-78.792,-177.536,10.754,149.515
C00518=1135.462,331.449,-78.759,-177.539,10.751,149.516
C00519=1135.466,331.202,-78.725,-177.543,10.749,149.516
C00520=1135.469,330.953,-78.691,-177.546,10.746,149.516
C00521=1135.473,330.706,-78.657,-177.549,10.743,149.516
C00522=1135.478,330.458,-78.624,-177.552,10.741,149.516
C00523=1135.482,330.211,-78.590,-177.555,10.739,149.517
C00524=1135.486,329.963,-78.556,-177.558,10.737,149.517
C00525=1135.490,329.715,-78.523,-177.561,10.734,149.517
C00526=1135.494,329.468,-78.489,-177.564,10.732,149.517
C00527=1135.498,329.220,-78.455,-177.568,10.729,149.518
C00528=1135.502,328.972,-78.421,-177.571,10.726,149.518
C00529=1135.506,328.724,-78.388,-177.574,10.724,149.518
C00530=1135.510,328.476,-78.355,-177.577,10.722,149.518
C00531=1135.514,328.229,-78.321,-177.581,10.719,149.518
C00532=1135.518,327.982,-78.288,-177.584,10.716,149.518
C00533=1135.521,327.733,-78.254,-177.587,10.714,149.519
C00534=1135.526,327.486,-78.220,-177.590,10.711,149.519
C00535=1135.530,327.238,-78.187,-177.593,10.709,149.519
C00536=1135.534,326.990,-78.154,-177.596,10.706,149.519
C00537=1135.538,326.743,-78.120,-177.600,10.704,149.519
C00538=1135.542,326.495,-78.086,-177.603,10.701,149.520
C00539=1135.546,326.247,-78.053,-177.606,10.699,149.520
C00540=1135.550,325.999,-78.020,-177.609,10.696,149.520
C00541=1135.554,325.752,-77.987,-177.613,10.694,149.520
C00542=1135.558,325.504,-77.953,-177.616,10.691,149.520
C00543=1135.562,325.256,-77.920,-177.619,10.688,149.521
C00544=1135.566,325.009,-77.886,-177.622,10.686,149.521
C00545=1135.570,324.761,-77.853,-177.625,10.683,149.521
C00546=1135.574,324.513,-77.820,-177.629,10.681,149.521
C00547=1135.578,324.265,-77.787,-177.632,10.678,149.521
C00548=1135.582,324.017,-77.753,-177.635,10.676,149.522
C00549=1135.586,323.770,-77.720,-177.638,10.673,149.522
C00550=1135.590,323.522,-77.687,-177.641,10.671,149.522
C00551=1135.595,323.274,-77.654,-177.645,10.668,149.522
C00552=1135.599,323.026,-77.621,-177.648,10.665,149.522
C00553=1135.603,322.779,-77.588,-177.651,10.663,149.523
C00554=1135.606,322.531,-77.555,-177.654,10.661,149.523
C00555=1135.610,322.283,-77.522,-177.657,10.658,149.523
C00556=1135.613,322.070,-77.493,-177.660,10.656,149.523
C00557=1135.617,321.856,-77.465,-177.662,10.654,149.523
C00558=1135.620,321.642,-77.436,-177.666,10.652,149.523
C00559=1135.624,321.429,-77.407,-177.668,10.650,149.524
C00560=1135.628,321.216,-77.379,-177.671,10.647,149.524
C00561=1135.631,321.002,-77.350,-177.673,10.645,149.524
C00562=1135.634,320.789,-77.322,-177.676,10.643,149.524
C00563=1135.638,320.575,-77.293,-177.679,10.641,149.524
C00564=1135.642,320.328,-77.260,-177.682,10.638,149.524
C00565=1135.646,320.080,-77.228,-177.685,10.636,149.525
C00566=1135.650,319.832,-77.195,-177.689,10.633,149.525
C00567=1135.654,319.584,-77.162,-177.692,10.630,149.525
C00568=1135.659,319.336,-77.129,-177.695,10.628,149.525
C00569=1135.663,319.089,-77.096,-177.698,10.626,149.525
C00570=1135.666,318.841,-77.063,-177.701,10.623,149.525
C00571=1135.670,318.593,-77.031,-177.704,10.620,149.526
C00572=1135.675,318.345,-76.998,-177.708,10.618,149.526
C00573=1135.679,318.097,-76.964,-177.710,10.616,149.526
C00574=1135.682,317.850,-76.932,-177.713,10.613,149.526
C00575=1135.687,317.602,-76.899,-177.717,10.611,149.527
C00576=1135.691,317.354,-76.866,-177.720,10.608,149.527
C00577=1135.695,317.106,-76.833,-177.723,10.606,149.527
C00578=1135.699,316.858,-76.801,-177.726,10.603,149.527
C00579=1135.703,316.610,-76.768,-177.729,10.601,149.527
C00580=1135.707,316.363,-76.735,-177.733,10.598,149.527
C00581=1135.711,316.115,-76.703,-177.736,10.595,149.528
C00582=1135.715,315.867,-76.670,-177.739,10.593,149.528
C00583=1135.719,315.619,-76.637,-177.742,10.591,149.528
C00584=1135.723,315.371,-76.605,-177.745,10.588,149.528
C00585=1135.727,315.123,-76.572,-177.748,10.585,149.528
C00586=1135.731,314.875,-76.539,-177.752,10.583,149.529
C00587=1135.735,314.628,-76.507,-177.755,10.580,149.529
C00588=1135.740,314.380,-76.475,-177.758,10.578,149.529
C00589=1135.743,314.133,-76.442,-177.761,10.575,149.529
C00590=1135.747,313.884,-76.410,-177.764,10.572,149.529
C00591=1135.752,313.636,-76.377,-177.768,10.570,149.530
C00592=1135.755,313.388,-76.345,-177.771,10.567,149.530
C00593=1135.759,313.141,-76.312,-177.774,10.565,149.530
C00594=1135.763,312.893,-76.280,-177.777,10.562,149.530
C00595=1135.767,312.645,-76.247,-177.780,10.560,149.530
C00596=1135.772,312.397,-76.215,-177.783,10.558,149.531
C00597=1135.776,312.149,-76.183,-177.786,10.555,149.531
C00598=1135.780,311.902,-76.150,-177.789,10.553,149.531
C00599=1135.784,311.653,-76.118,-177.792,10.550,149.531
C00600=1135.788,311.406,-76.085,-177.795,10.548,149.531
C00601=1135.792,311.158,-76.053,-177.799,10.545,149.531
C00602=1135.797,310.910,-76.021,-177.802,10.542,149.532
C00603=1135.800,310.663,-75.988,-177.805,10.540,149.532
C00604=1135.805,310.414,-75.956,-177.808,10.537,149.532
C00605=1135.808,310.166,-75.924,-177.811,10.535,149.532
C00606=1135.813,309.918,-75.891,-177.815,10.532,149.532
C00607=1135.816,309.670,-75.859,-177.817,10.529,149.532
C00608=1135.821,309.423,-75.827,-177.821,10.527,149.533
C00609=1135.825,309.175,-75.795,-177.824,10.524,149.533
C00610=1135.829,308.927,-75.763,-177.827,10.522,149.533
C00611=1135.833,308.679,-75.730,-177.830,10.519,149.533
C00612=1135.837,308.454,-75.701,-177.833,10.517,149.533
C00613=1135.840,308.229,-75.672,-177.836,10.515,149.534
C00614=1135.844,308.004,-75.643,-177.839,10.512,149.534
C00615=1135.847,307.779,-75.614,-177.841,10.510,149.534
C00616=1135.852,307.555,-75.585,-177.845,10.508,149.534
C00617=1135.856,307.329,-75.555,-177.847,10.506,149.534
C00618=1135.860,307.104,-75.527,-177.850,10.503,149.534
C00619=1135.863,306.879,-75.497,-177.853,10.501,149.535
C00620=1135.867,306.631,-75.465,-177.855,10.499,149.535
C00621=1135.871,306.384,-75.434,-177.859,10.496,149.535
C00622=1135.875,306.136,-75.401,-177.862,10.494,149.535
C00623=1135.879,305.888,-75.369,-177.865,10.491,149.535
C00624=1135.883,305.640,-75.338,-177.868,10.489,149.536
C00625=1135.888,305.392,-75.306,-177.871,10.486,149.536
C00626=1135.892,305.144,-75.274,-177.875,10.483,149.536
C00627=1135.895,304.896,-75.242,-177.878,10.481,149.536
C00628=1135.900,304.648,-75.210,-177.881,10.478,149.536
C00629=1135.904,304.400,-75.178,-177.884,10.475,149.536
C00630=1135.908,304.152,-75.146,-177.887,10.473,149.537
C00631=1135.912,303.905,-75.115,-177.891,10.471,149.537
C00632=1135.917,303.657,-75.082,-177.893,10.468,149.537
C00633=1135.920,303.409,-75.050,-177.897,10.465,149.537
C00634=1135.925,303.161,-75.019,-177.900,10.463,149.537
C00635=1135.929,302.913,-74.988,-177.903,10.460,149.538
C00636=1135.933,302.664,-74.955,-177.905,10.458,149.538
C00637=1135.937,302.417,-74.924,-177.909,10.456,149.538
C00638=1135.941,302.169,-74.892,-177.912,10.453,149.538
C00639=1135.945,301.921,-74.860,-177.915,10.451,149.538
C00640=1135.949,301.673,-74.829,-177.918,10.448,149.538
C00641=1135.954,301.424,-74.797,-177.921,10.445,149.539
C00642=1135.958,301.177,-74.765,-177.924,10.443,149.539
C00643=1135.962,300.929,-74.734,-177.927,10.440,149.539
C00644=1135.966,300.682,-74.702,-177.931,10.438,149.539
C00645=1135.970,300.433,-74.671,-177.934,10.435,149.539
C00646=1135.974,300.185,-74.639,-177.937,10.432,149.540
C00647=1135.978,299.938,-74.608,-177.940,10.430,149.540
C00648=1135.983,299.689,-74.576,-177.943,10.427,149.540
C00649=1135.987,299.441,-74.544,-177.946,10.425,149.540
C00650=1135.991,299.193,-74.513,-177.950,10.422,149.540
C00651=1135.996,298.945,-74.482,-177.953,10.419,149.540
C00652=1135.999,298.697,-74.450,-177.955,10.418,149.541
C00653=1136.003,298.449,-74.418,-177.958,10.415,149.541
C00654=1136.008,298.201,-74.387,-177.962,10.412,149.541
C00655=1136.011,297.953,-74.356,-177.964,10.410,149.541
C00656=1136.016,297.705,-74.325,-177.968,10.407,149.541
C00657=1136.020,297.457,-74.293,-177.971,10.405,149.541
C00658=1136.024,297.209,-74.262,-177.974,10.402,149.542
C00659=1136.028,296.961,-74.230,-177.977,10.399,149.542
C00660=1136.032,296.714,-74.199,-177.980,10.397,149.542
C00661=1136.036,296.465,-74.168,-177.983,10.394,149.542
C00662=1136.041,296.218,-74.136,-177.987,10.392,149.542
C00663=1136.045,295.969,-74.105,-177.990,10.389,149.543
C00664=1136.066,294.691,-73.943,-177.108,8.658,148.873
C00665=1136.070,294.443,-73.913,-177.111,8.654,148.872
C00666=1136.074,294.195,-73.882,-177.114,8.650,148.872
C00667=1136.079,293.947,-73.851,-177.116,8.648,148.872
C00668=1136.082,293.699,-73.821,-177.119,8.643,148.872
C00669=1136.087,293.451,-73.790,-177.122,8.641,148.872
C00670=1136.091,293.203,-73.759,-177.124,8.637,148.872
C00671=1136.095,292.954,-73.729,-177.127,8.633,148.872
C00672=1136.099,292.706,-73.698,-177.130,8.630,148.872
C00673=1136.104,292.458,-73.667,-177.133,8.626,148.872
C00674=1136.107,292.210,-73.637,-177.135,8.623,148.871
C00675=1136.112,291.962,-73.606,-177.138,8.620,148.872
C00676=1136.116,291.714,-73.575,-177.141,8.616,148.871
C00677=1136.120,291.466,-73.545,-177.144,8.613,148.871
C00678=1136.124,291.218,-73.514,-177.146,8.610,148.871
C00679=1136.129,290.969,-73.484,-177.149,8.606,148.871
C00680=1136.133,290.722,-73.454,-177.152,8.603,148.871
C00681=1136.137,290.473,-73.422,-177.154,8.600,148.871
C00682=1136.141,290.225,-73.392,-177.157,8.596,148.871
C00683=1136.146,289.977,-73.361,-177.160,8.593,148.871
C00684=1136.149,289.730,-73.331,-177.162,8.589,148.871
C00685=1136.154,289.480,-73.301,-177.166,8.586,148.871
C00686=1136.158,289.233,-73.271,-177.168,8.582,148.870
C00687=1136.162,288.985,-73.240,-177.171,8.579,148.870
C00688=1136.167,288.737,-73.209,-177.174,8.575,148.870
C00689=1136.171,288.489,-73.179,-177.176,8.572,148.870
C00690=1136.175,288.240,-73.149,-177.179,8.569,148.870
C00691=1136.179,287.992,-73.118,-177.182,8.565,148.870
C00692=1136.184,287.744,-73.088,-177.185,8.562,148.870
C00693=1136.188,287.468,-73.055,-177.188,8.558,148.870
C00694=1136.193,287.193,-73.021,-177.191,8.554,148.870
C00695=1136.197,286.918,-72.987,-177.193,8.551,148.870
C00696=1136.202,286.641,-72.954,-177.197,8.547,148.870
C00697=1136.206,286.394,-72.923,-177.200,8.543,148.869
C00698=1136.210,286.146,-72.893,-177.202,8.540,148.869
C00699=1136.215,285.897,-72.863,-177.205,8.537,148.869
C00700=1136.218,285.649,-72.833,-177.208,8.533,148.869
C00701=1136.223,285.400,-72.803,-177.211,8.530,148.869
C00702=1136.227,285.153,-72.772,-177.213,8.527,148.869
C00703=1136.231,284.904,-72.743,-177.216,8.524,148.869
C00704=1136.236,284.657,-72.712,-177.219,8.520,148.869
C00705=1136.240,284.408,-72.683,-177.221,8.517,148.869
C00706=1136.245,284.160,-72.652,-177.224,8.514,148.869
C00707=1136.249,283.912,-72.623,-177.227,8.510,148.869
C00708=1136.253,283.664,-72.592,-177.229,8.507,148.869
C00709=1136.257,283.415,-72.562,-177.232,8.504,148.869
C00710=1136.261,283.167,-72.532,-177.235,8.500,148.868
C00711=1136.265,282.919,-72.502,-177.238,8.497,148.868
C00712=1136.270,282.671,-72.472,-177.240,8.494,148.868
C00713=1136.274,282.423,-72.442,-177.243,8.491,148.868
C00714=1136.278,282.175,-72.413,-177.246,8.487,148.868
C00715=1136.282,281.927,-72.382,-177.249,8.484,148.868
C00716=1136.287,281.678,-72.352,-177.252,8.481,148.868
C00717=1136.291,281.430,-72.323,-177.255,8.477,148.868
C00718=1136.295,281.183,-72.293,-177.257,8.474,148.868
C00719=1136.299,280.934,-72.263,-177.260,8.471,148.868
C00720=1136.304,280.686,-72.233,-177.262,8.468,148.868
C00721=1136.308,280.438,-72.203,-177.265,8.464,148.868
C00722=1136.312,280.190,-72.174,-177.268,8.461,148.868
C00723=1136.316,279.942,-72.144,-177.271,8.457,148.868
C00724=1136.321,279.693,-72.114,-177.274,8.454,148.868
C00725=1136.325,279.445,-72.084,-177.276,8.450,148.868
C00726=1136.329,279.197,-72.055,-177.279,8.447,148.868
C00727=1136.333,278.949,-72.025,-177.282,8.445,148.868
C00728=1136.338,278.701,-71.996,-177.285,8.440,148.867
C00729=1136.342,278.452,-71.966,-177.288,8.438,148.868
C00730=1136.346,278.204,-71.937,-177.290,8.434,148.867
C00731=1136.351,277.956,-71.906,-177.293,8.431,148.867
C00732=1136.355,277.708,-71.877,-177.296,8.427,148.867
C00733=1136.359,277.459,-71.847,-177.298,8.424,148.867
C00734=1136.363,277.211,-71.818,-177.301,8.421,148.867
C00735=1136.367,276.963,-71.788,-177.304,8.418,148.867
C00736=1136.372,276.715,-71.759,-177.307,8.414,148.867
C00737=1136.376,276.466,-71.729,-177.309,8.411,148.867
C00738=1136.380,276.218,-71.700,-177.312,8.408,148.867
C00739=1136.384,275.970,-71.670,-177.314,8.405,148.867
C00740=1136.388,275.722,-71.641,-177.318,8.401,148.867
C00741=1136.392,275.473,-71.611,-177.321,8.398,148.867
C00742=1136.397,275.225,-71.582,-177.323,8.395,148.867
C00743=1136.401,274.977,-71.553,-177.326,8.392,148.867
C00744=1136.406,274.729,-71.523,-177.329,8.388,148.867
C00745=1136.410,274.481,-71.494,-177.332,8.385,148.867
C00746=1136.414,274.233,-71.465,-177.334,8.382,148.867
C00747=1136.418,273.984,-71.435,-177.337,8.379,148.867
C00748=1136.422,273.736,-71.406,-177.339,8.376,148.867
C00749=1136.427,273.488,-71.376,-177.343,8.372,148.867
C00750=1136.431,273.240,-71.347,-177.345,8.369,148.867
C00751=1136.435,272.991,-71.318,-177.348,8.366,148.867
C00752=1136.439,272.742,-71.289,-177.351,8.363,148.867
C00753=1136.444,272.495,-71.259,-177.354,8.359,148.866
C00754=1136.448,272.247,-71.230,-177.356,8.356,148.867
C00755=1136.452,271.998,-71.201,-177.359,8.353,148.866
C00756=1136.457,271.749,-71.172,-177.362,8.350,148.866
C00757=1136.461,271.501,-71.142,-177.364,8.347,148.867
C00758=1136.465,271.253,-71.113,-177.367,8.343,148.866
C00759=1136.469,271.006,-71.084,-177.370,8.340,148.866
C00760=1136.474,270.757,-71.056,-177.373,8.337,148.866
C00761=1136.478,270.509,-71.026,-177.375,8.334,148.866
C00762=1136.482,270.260,-70.997,-177.379,8.330,148.866
C00763=1136.486,270.012,-70.967,-177.381,8.327,148.866
C00764=1136.492,269.764,-70.939,-177.384,8.324,148.866
C00765=1136.495,269.516,-70.910,-177.387,8.321,148.866
C00766=1136.499,269.268,-70.881,-177.389,8.318,148.866
C00767=1136.504,269.019,-70.852,-177.392,8.314,148.866
C00768=1136.508,268.771,-70.823,-177.395,8.311,148.866
C00769=1136.513,268.522,-70.794,-177.398,8.308,148.866
C00770=1136.516,268.274,-70.765,-177.400,8.305,148.866
C00771=1136.521,268.025,-70.736,-177.403,8.302,148.866
C00772=1136.526,267.778,-70.707,-177.406,8.299,148.866
C00773=1136.530,267.530,-70.678,-177.409,8.296,148.866
C00774=1136.534,267.281,-70.650,-177.412,8.292,148.866
C00775=1136.538,267.033,-70.620,-177.414,8.289,148.866
C00776=1136.543,266.785,-70.592,-177.417,8.287,148.866
C00777=1136.547,266.536,-70.562,-177.420,8.283,148.866
C00778=1136.551,266.288,-70.534,-177.423,8.280,148.866
C00779=1136.555,266.039,-70.505,-177.426,8.277,148.866
C00780=1136.560,265.791,-70.477,-177.428,8.273,148.866
C00781=1136.564,265.543,-70.448,-177.431,8.270,148.866
C00782=1136.568,265.294,-70.419,-177.434,8.268,148.866
C00783=1136.573,265.046,-70.391,-177.436,8.265,148.866
C00784=1136.576,264.798,-70.362,-177.439,8.261,148.866
C00785=1136.581,264.549,-70.333,-177.442,8.258,148.866
C00786=1136.586,264.301,-70.305,-177.445,8.255,148.866
C00787=1136.589,264.053,-70.276,-177.448,8.252,148.866
C00788=1136.594,263.804,-70.247,-177.450,8.249,148.866
C00789=1136.599,263.556,-70.219,-177.453,8.246,148.866
C00790=1136.603,263.308,-70.190,-177.456,8.242,148.866
C00791=1136.608,263.060,-70.161,-177.459,8.239,148.866
C00792=1136.611,262.811,-70.133,-177.461,8.236,148.866
C00793=1136.616,262.563,-70.105,-177.464,8.233,148.866
C00794=1136.620,262.315,-70.076,-177.467,8.230,148.866
C00795=1136.624,262.066,-70.047,-177.470,8.227,148.866
C00796=1136.629,261.818,-70.019,-177.473,8.223,148.866
C00797=1136.634,261.544,-69.988,-177.476,8.220,148.866
C00798=1136.639,261.271,-69.956,-177.479,8.216,148.866
C00799=1136.643,260.997,-69.925,-177.482,8.213,148.866
C00800=1136.648,260.723,-69.894,-177.485,8.210,148.866
C00801=1136.652,260.475,-69.865,-177.487,8.206,148.866
C00802=1136.657,260.227,-69.837,-177.490,8.203,148.866
C00803=1136.660,259.979,-69.808,-177.493,8.201,148.866
C00804=1136.665,259.731,-69.780,-177.496,8.198,148.866
C00805=1136.669,259.482,-69.752,-177.499,8.194,148.866
C00806=1136.674,259.233,-69.723,-177.502,8.191,148.866
C00807=1136.678,258.985,-69.695,-177.504,8.188,148.866
C00808=1136.682,258.737,-69.667,-177.507,8.185,148.866
C00809=1136.687,258.488,-69.639,-177.510,8.182,148.866
C00810=1136.691,258.240,-69.610,-177.513,8.179,148.866
C00811=1136.696,257.992,-69.582,-177.515,8.176,148.866
C00812=1136.699,257.743,-69.554,-177.518,8.173,148.866
C00813=1136.704,257.495,-69.526,-177.521,8.169,148.866
C00814=1136.708,257.246,-69.497,-177.524,8.166,148.866
C00815=1136.713,256.998,-69.470,-177.527,8.163,148.867
C00816=1136.716,256.750,-69.442,-177.529,8.160,148.866
C00817=1136.722,256.502,-69.413,-177.532,8.157,148.866
C00818=1136.725,256.253,-69.385,-177.535,8.154,148.867
C00819=1136.730,256.005,-69.357,-177.538,8.151,148.867
C00820=1136.734,255.756,-69.329,-177.540,8.148,148.867
C00821=1136.739,255.508,-69.301,-177.543,8.145,148.867
C00822=1136.743,255.259,-69.273,-177.546,8.141,148.867
C00823=1136.748,255.011,-69.245,-177.549,8.138,148.867
C00824=1136.751,254.763,-69.217,-177.552,8.136,148.867
C00825=1136.756,254.515,-69.189,-177.555,8.133,148.867
C00826=1136.761,254.266,-69.161,-177.557,8.130,148.867
C00827=1136.765,254.017,-69.133,-177.560,8.127,148.867
C00828=1136.769,253.769,-69.105,-177.563,8.124,148.867
C00829=1136.773,253.521,-69.077,-177.565,8.121,148.867
C00830=1136.778,253.272,-69.050,-177.568,8.118,148.867
C00831=1136.782,253.023,-69.022,-177.571,8.115,148.867
C00832=1136.786,252.776,-68.994,-177.574,8.111,148.867
C00833=1136.791,252.528,-68.966,-177.577,8.108,148.867
C00834=1136.795,252.278,-68.939,-177.579,8.105,148.867
C00835=1136.800,252.030,-68.910,-177.582,8.102,148.867
C00836=1136.804,251.782,-68.882,-177.585,8.099,148.867
C00837=1136.808,251.533,-68.855,-177.588,8.096,148.867
C00838=1136.813,251.285,-68.827,-177.591,8.093,148.867
C00839=1136.817,251.036,-68.800,-177.593,8.090,148.867
C00840=1136.821,250.788,-68.772,-177.596,8.087,148.867
C00841=1136.825,250.540,-68.744,-177.599,8.085,148.867
C00842=1136.830,250.291,-68.716,-177.601,8.081,148.867
C00843=1136.835,250.043,-68.688,-177.604,8.078,148.867
C00844=1136.839,249.795,-68.661,-177.607,8.075,148.867
C00845=1136.843,249.546,-68.633,-177.610,8.072,148.868
C00846=1136.848,249.297,-68.606,-177.613,8.069,148.868
C00847=1136.852,249.050,-68.578,-177.616,8.066,148.868
C00848=1136.856,248.800,-68.551,-177.619,8.063,148.868
C00849=1136.860,248.553,-68.523,-177.622,8.060,148.868
C00850=1136.865,248.304,-68.496,-177.624,8.057,148.868
C00851=1136.869,248.055,-68.468,-177.627,8.054,148.868
C00852=1136.873,247.807,-68.441,-177.630,8.051,148.868
C00853=1136.878,247.559,-68.413,-177.632,8.048,148.868
C00854=1136.882,247.310,-68.386,-177.635,8.045,148.868
C00855=1136.887,247.061,-68.359,-177.638,8.042,148.868
C00856=1136.891,246.814,-68.331,-177.641,8.039,148.868
C00857=1136.896,246.565,-68.304,-177.644,8.036,148.868
C00858=1136.899,246.316,-68.276,-177.646,8.034,148.868
C00859=1136.904,246.068,-68.249,-177.649,8.031,148.868
C00860=1136.909,245.819,-68.222,-177.652,8.028,148.868
C00861=1136.913,245.572,-68.194,-177.655,8.025,148.869
C00862=1136.917,245.322,-68.166,-177.658,8.022,148.869
C00863=1136.922,245.074,-68.139,-177.660,8.019,148.868
C00864=1136.926,244.825,-68.112,-177.663,8.016,148.869
C00865=1136.931,244.578,-68.084,-177.666,8.012,148.869
C00866=1136.935,244.328,-68.057,-177.669,8.009,148.869
C00867=1136.939,244.080,-68.030,-177.672,8.006,148.869
C00868=1136.944,243.831,-68.003,-177.674,8.003,148.869
C00869=1136.948,243.583,-67.975,-177.677,8.000,148.869
C00870=1136.952,243.335,-67.949,-177.680,7.997,148.869
C00871=1136.956,243.086,-67.921,-177.683,7.995,148.869
C00872=1136.961,242.838,-67.894,-177.686,7.992,148.869
C00873=1136.966,242.589,-67.867,-177.688,7.989,148.869
C00874=1136.970,242.341,-67.840,-177.691,7.986,148.869
C00875=1136.975,242.092,-67.813,-177.694,7.983,148.869
C00876=1136.979,241.843,-67.785,-177.697,7.980,148.869
C00877=1136.983,241.595,-67.758,-177.700,7.977,148.870
C00878=1136.987,241.347,-67.731,-177.702,7.974,148.870
C00879=1136.992,241.098,-67.704,-177.705,7.971,148.870
C00880=1136.997,240.850,-67.677,-177.708,7.968,148.870
C00881=1137.001,240.602,-67.651,-177.711,7.965,148.870
C00882=1137.005,240.353,-67.624,-177.714,7.963,148.870
C00883=1137.009,240.104,-67.596,-177.716,7.960,148.870
C00884=1137.014,239.855,-67.569,-177.719,7.957,148.870
C00885=1137.019,239.607,-67.542,-177.722,7.953,148.870
C00886=1137.022,239.359,-67.516,-177.724,7.951,148.870
C00887=1137.027,239.110,-67.489,-177.727,7.948,148.870
C00888=1137.032,238.862,-67.461,-177.730,7.945,148.870
C00889=1137.036,238.614,-67.435,-177.733,7.942,148.870
C00890=1137.040,238.365,-67.408,-177.736,7.939,148.870
C00891=1137.045,238.117,-67.381,-177.738,7.936,148.870
C00892=1137.049,237.868,-67.355,-177.741,7.933,148.871
C00893=1137.053,237.619,-67.328,-177.744,7.930,148.871
C00894=1137.058,237.370,-67.301,-177.747,7.927,148.871
C00895=1137.062,237.122,-67.274,-177.750,7.924,148.871
C00896=1137.067,236.873,-67.247,-177.752,7.921,148.871
C00897=1137.071,236.625,-67.220,-177.755,7.919,148.871
C00898=1137.075,236.376,-67.194,-177.758,7.916,148.871
C00899=1137.080,236.128,-67.167,-177.761,7.913,148.871
C00900=1137.085,235.879,-67.140,-177.764,7.910,148.871
C00901=1137.089,235.608,-67.111,-177.767,7.907,148.871
C00902=1137.094,235.336,-67.082,-177.770,7.904,148.872
C00903=1137.099,235.063,-67.053,-177.773,7.901,148.872
C00904=1137.104,234.792,-67.024,-177.776,7.898,148.872
C00905=1137.108,234.544,-66.997,-177.779,7.895,148.872
C00906=1137.113,234.294,-66.971,-177.782,7.892,148.872
C00907=1137.117,234.046,-66.944,-177.784,7.889,148.872
C00908=1137.122,233.798,-66.917,-177.787,7.886,148.872
C00909=1137.126,233.549,-66.892,-177.790,7.883,148.872
C00910=1137.131,233.300,-66.865,-177.793,7.880,148.872
C00911=1137.134,233.052,-66.838,-177.796,7.877,148.872
C00912=1137.139,232.803,-66.812,-177.798,7.874,148.872
C00913=1137.143,232.555,-66.785,-177.801,7.872,148.872
C00914=1137.148,232.306,-66.759,-177.804,7.869,148.873
C00915=1137.152,232.058,-66.732,-177.807,7.866,148.873
C00916=1137.157,231.809,-66.705,-177.809,7.864,148.873
C00917=1137.161,231.560,-66.680,-177.812,7.861,148.873
C00918=1137.166,231.312,-66.653,-177.815,7.858,148.873
C00919=1137.170,231.063,-66.627,-177.818,7.855,148.873
C00920=1137.175,230.815,-66.600,-177.821,7.852,148.873
C00921=1137.179,230.566,-66.574,-177.823,7.849,148.873
C00922=1137.183,230.318,-66.548,-177.826,7.847,148.873
C00923=1137.188,230.069,-66.522,-177.829,7.844,148.874
C00924=1137.192,229.821,-66.495,-177.832,7.841,148.874
C00925=1137.197,229.572,-66.469,-177.835,7.838,148.874
C00926=1137.201,229.323,-66.443,-177.838,7.835,148.874
C00927=1137.205,229.075,-66.417,-177.840,7.832,148.874
C00928=1137.210,228.826,-66.390,-177.843,7.829,148.874
C00929=1137.214,228.578,-66.364,-177.846,7.826,148.874
C00930=1137.218,228.329,-66.338,-177.849,7.824,148.874
C00931=1137.224,228.080,-66.312,-177.851,7.822,148.875
C00932=1137.228,227.832,-66.286,-177.854,7.819,148.875
C00933=1137.232,227.583,-66.260,-177.857,7.816,148.875
C00934=1137.237,227.334,-66.233,-177.860,7.813,148.875
C00935=1137.241,227.086,-66.207,-177.863,7.810,148.875
C00936=1137.245,226.837,-66.181,-177.865,7.807,148.875
C00937=1137.250,226.588,-66.155,-177.868,7.804,148.875
C00938=1137.255,226.340,-66.130,-177.871,7.801,148.875
C00939=1137.259,226.092,-66.103,-177.874,7.798,148.875
C00940=1137.263,225.843,-66.077,-177.877,7.796,148.876
C00941=1137.268,225.594,-66.051,-177.880,7.793,148.876
C00942=1137.272,225.345,-66.025,-177.882,7.791,148.876
C00943=1137.277,225.098,-65.999,-177.885,7.788,148.876
C00944=1137.281,224.849,-65.973,-177.888,7.785,148.876
C00945=1137.285,224.600,-65.948,-177.891,7.782,148.876
C00946=1137.290,224.351,-65.921,-177.893,7.779,148.876
C00947=1137.295,224.102,-65.895,-177.896,7.776,148.876
C00948=1137.299,223.854,-65.870,-177.899,7.774,148.877
C00949=1137.304,223.605,-65.844,-177.902,7.771,148.877
C00950=1137.308,223.357,-65.818,-177.905,7.768,148.877
C00951=1137.313,223.108,-65.792,-177.907,7.766,148.877
C00952=1137.317,222.860,-65.766,-177.910,7.763,148.877
C00953=1137.322,222.611,-65.740,-177.913,7.760,148.877
C00954=1137.326,222.362,-65.715,-177.916,7.757,148.877
C00955=1137.330,222.113,-65.689,-177.919,7.754,148.877
C00956=1137.335,221.865,-65.664,-177.922,7.752,148.878
C00957=1137.339,221.616,-65.638,-177.925,7.749,148.878
C00958=1137.343,221.368,-65.612,-177.927,7.746,148.878
C00959=1137.348,221.120,-65.587,-177.930,7.743,148.878
C00960=1137.353,220.870,-65.560,-177.932,7.741,148.878
C00961=1137.357,220.622,-65.535,-177.936,7.738,148.878
C00962=1137.362,220.374,-65.509,-177.939,7.735,148.878
C00963=1137.366,220.125,-65.483,-177.941,7.732,148.878
C00964=1137.371,219.876,-65.458,-177.944,7.729,148.879
C00965=1137.375,219.627,-65.433,-177.947,7.727,148.879
C00966=1137.380,219.378,-65.407,-177.950,7.724,148.879
C00967=1137.384,219.130,-65.381,-177.952,7.722,148.879
C00968=1137.388,218.881,-65.356,-177.955,7.719,148.879
C00969=1137.393,218.633,-65.330,-177.958,7.716,148.879
C00970=1137.397,218.384,-65.305,-177.961,7.713,148.879
C00971=1137.402,218.135,-65.279,-177.964,7.710,148.879
C00972=1137.407,217.886,-65.254,-177.967,7.708,148.880
C00973=1137.411,217.638,-65.228,-177.969,7.706,148.880
C00974=1137.416,217.389,-65.203,-177.972,7.703,148.880
C00975=1137.420,217.141,-65.177,-177.975,7.700,148.880
C00976=1137.424,216.892,-65.152,-177.978,7.697,148.880
C00977=1137.429,216.643,-65.127,-177.981,7.694,148.880
C00978=1137.433,216.395,-65.102,-177.984,7.691,148.881
C00979=1137.437,216.146,-65.076,-177.986,7.689,148.881
C00980=1137.442,215.897,-65.051,-177.989,7.686,148.881
C00981=1137.446,215.648,-65.026,-177.992,7.684,148.881
C00982=1137.451,215.400,-65.000,-177.995,7.681,148.881
C00983=1137.456,215.151,-64.975,-177.998,7.678,148.881
C00984=1137.461,214.903,-64.950,-178.000,7.675,148.881
C00985=1137.465,214.654,-64.924,-178.003,7.673,148.882
C00986=1137.469,214.405,-64.900,-178.006,7.671,148.882
C00987=1137.474,214.157,-64.874,-178.009,7.668,148.882
C00988=1137.478,213.908,-64.848,-178.012,7.665,148.882
C00989=1137.483,213.659,-64.824,-178.014,7.662,148.882
C00990=1137.487,213.410,-64.798,-178.018,7.659,148.882
C00991=1137.491,213.162,-64.774,-178.020,7.657,148.883
C00992=1137.496,212.913,-64.748,-178.023,7.654,148.883
C00993=1137.501,212.664,-64.723,-178.025,7.651,148.883
C00994=1137.505,212.416,-64.698,-178.029,7.649,148.883
C00995=1137.510,212.167,-64.673,-178.032,7.646,148.883
C00996=1137.514,211.918,-64.648,-178.034,7.644,148.883
C00997=1137.519,211.670,-64.623,-178.037,7.641,148.883
C00998=1137.523,211.421,-64.598,-178.040,7.638,148.884
C00999=1137.528,211.172,-64.573,-178.043,7.636,148.884
C01000=1137.532,210.924,-64.548,-178.045,7.633,148.884
C01001=1137.537,210.675,-64.523,-178.048,7.631,148.884
C01002=1137.541,210.426,-64.497,-178.051,7.628,148.884
C01003=1137.546,210.177,-64.473,-178.054,7.625,148.885
C01004=1137.550,209.928,-64.448,-178.057,7.622,148.885
C01005=1137.555,209.658,-64.421,-178.060,7.620,148.885
C01006=1137.560,209.387,-64.394,-178.063,7.617,148.885
C01007=1137.565,209.117,-64.366,-178.065,7.614,148.885
C01008=1137.570,208.846,-64.339,-178.069,7.611,148.885
C01009=1137.574,208.597,-64.314,-178.072,7.608,148.886
C01010=1137.579,208.349,-64.290,-178.074,7.605,148.886
C01011=1137.584,208.100,-64.265,-178.077,7.604,148.886
C01012=1137.588,207.851,-64.240,-178.080,7.601,148.886
C01013=1137.592,207.603,-64.216,-178.083,7.598,148.886
C01014=1137.597,207.353,-64.191,-178.086,7.595,148.887
C01015=1137.601,207.105,-64.167,-178.088,7.593,148.887
C01016=1137.606,206.856,-64.141,-178.091,7.590,148.887
C01017=1137.611,206.607,-64.116,-178.094,7.588,148.887
C01018=1137.615,206.359,-64.092,-178.097,7.585,148.887
C01019=1137.620,206.109,-64.067,-178.100,7.582,148.887
C01020=1137.624,205.861,-64.043,-178.103,7.580,148.888
C01021=1137.629,205.613,-64.018,-178.105,7.577,148.888
C01022=1137.633,205.364,-63.993,-178.108,7.575,148.888
C01023=1137.638,205.115,-63.968,-178.111,7.573,148.888
C01024=1137.642,204.867,-63.944,-178.114,7.570,148.888
C01025=1137.647,204.617,-63.919,-178.117,7.567,148.888
C01026=1137.652,204.369,-63.895,-178.120,7.564,148.889
C01027=1137.656,204.120,-63.871,-178.122,7.562,148.889
C01028=1137.661,203.871,-63.846,-178.125,7.559,148.889
C01029=1137.665,203.622,-63.821,-178.128,7.557,148.889
C01030=1137.670,203.374,-63.797,-178.131,7.554,148.889
C01031=1137.674,203.125,-63.772,-178.133,7.552,148.890
C01032=1137.678,202.877,-63.748,-178.136,7.549,148.890
C01033=1137.683,202.628,-63.723,-178.139,7.546,148.890
C01034=1137.687,202.379,-63.698,-178.142,7.544,148.890
C01035=1137.692,202.130,-63.674,-178.145,7.542,148.890
C01036=1137.697,201.881,-63.650,-178.148,7.539,148.891
C01037=1137.701,201.632,-63.626,-178.150,7.536,148.891
C01038=1137.706,201.383,-63.601,-178.153,7.534,148.891
C01039=1137.710,201.135,-63.577,-178.156,7.531,148.891
C01040=1137.715,200.886,-63.553,-178.159,7.529,148.892
C01041=1137.719,200.637,-63.528,-178.162,7.526,148.892
C01042=1137.724,200.389,-63.504,-178.164,7.524,148.892
C01043=1137.729,200.140,-63.479,-178.167,7.521,148.892
C01044=1137.733,199.891,-63.455,-178.170,7.518,148.892
C01045=1137.737,199.642,-63.431,-178.173,7.517,148.893
C01046=1137.742,199.393,-63.407,-178.176,7.514,148.893
C01047=1137.747,199.145,-63.383,-178.179,7.511,148.893
C01048=1137.751,198.896,-63.359,-178.181,7.509,148.893
C01049=1137.756,198.647,-63.334,-178.184,7.506,148.893
C01050=1137.760,198.398,-63.310,-178.187,7.504,148.894
C01051=1137.765,198.149,-63.286,-178.190,7.501,148.894
C01052=1137.769,197.901,-63.262,-178.192,7.499,148.894
C01053=1137.774,197.652,-63.238,-178.196,7.496,148.894
C01054=1137.778,197.403,-63.213,-178.199,7.493,148.894
C01055=1137.783,197.154,-63.190,-178.201,7.492,148.895
C01056=1137.787,196.906,-63.166,-178.204,7.489,148.895
C01057=1137.792,196.657,-63.141,-178.207,7.486,148.895
C01058=1137.797,196.408,-63.117,-178.210,7.484,148.895
C01059=1137.801,196.159,-63.093,-178.212,7.481,148.895
C01060=1137.805,195.910,-63.069,-178.216,7.479,148.896
C01061=1137.811,195.661,-63.045,-178.218,7.477,148.896
C01062=1137.815,195.413,-63.021,-178.221,7.474,148.896
C01063=1137.819,195.164,-62.997,-178.224,7.471,148.896
C01064=1137.824,194.915,-62.974,-178.226,7.469,148.896
C01065=1137.829,194.667,-62.950,-178.229,7.466,148.897
C01066=1137.832,194.418,-62.925,-178.232,7.464,148.897
C01067=1137.838,194.168,-62.901,-178.235,7.462,148.897
C01068=1137.842,193.920,-62.877,-178.238,7.459,148.897
C01069=1137.847,193.671,-62.854,-178.241,7.456,148.898
C01070=1137.851,193.422,-62.830,-178.243,7.454,148.898
C01071=1137.856,193.173,-62.806,-178.247,7.452,148.898
C01072=1137.860,192.925,-62.782,-178.249,7.450,148.898
C01073=1137.865,192.676,-62.759,-178.252,7.447,148.898
C01074=1137.869,192.428,-62.735,-178.255,7.444,148.899
C01075=1137.875,192.178,-62.711,-178.257,7.442,148.899
C01076=1137.879,191.930,-62.687,-178.260,7.440,148.899
C01077=1137.883,191.680,-62.663,-178.263,7.437,148.899
C01078=1137.888,191.431,-62.640,-178.266,7.435,148.900
C01079=1137.892,191.183,-62.616,-178.269,7.432,148.900
C01080=1137.897,190.934,-62.592,-178.272,7.430,148.900
C01081=1137.902,190.685,-62.568,-178.274,7.427,148.900
C01082=1137.906,190.436,-62.545,-178.278,7.425,148.901
C01083=1137.911,190.187,-62.522,-178.280,7.423,148.901
C01084=1137.915,189.939,-62.497,-178.283,7.420,148.901
C01085=1137.920,189.690,-62.474,-178.286,7.417,148.901
C01086=1137.925,189.441,-62.451,-178.289,7.416,148.901
C01087=1137.929,189.192,-62.427,-178.291,7.413,148.902
C01088=1137.934,188.943,-62.403,-178.295,7.410,148.902
C01089=1137.939,188.694,-62.380,-178.297,7.408,148.902
C01090=1137.943,188.446,-62.356,-178.300,7.406,148.902
C01091=1137.948,188.197,-62.332,-178.302,7.404,148.903
C01092=1137.952,187.948,-62.309,-178.306,7.401,148.903
C01093=1137.957,187.699,-62.286,-178.309,7.398,148.903
C01094=1137.961,187.450,-62.262,-178.311,7.396,148.903
C01095=1137.966,187.201,-62.238,-178.314,7.394,148.903
C01096=1137.971,186.952,-62.215,-178.317,7.392,148.904
C01097=1137.975,186.703,-62.192,-178.320,7.389,148.904
C01098=1137.979,186.454,-62.169,-178.323,7.386,148.904
C01099=1137.984,186.206,-62.145,-178.325,7.384,148.904
C01100=1137.989,185.957,-62.121,-178.328,7.382,148.905
C01101=1137.993,185.708,-62.098,-178.331,7.380,148.905
C01102=1137.999,185.460,-62.075,-178.334,7.377,148.905
C01103=1138.003,185.211,-62.052,-178.336,7.375,148.905
C01104=1138.008,184.962,-62.028,-178.339,7.372,148.906
C01105=1138.012,184.713,-62.006,-178.342,7.370,148.906
C01106=1138.017,184.464,-61.982,-178.345,7.368,148.906
C01107=1138.021,184.215,-61.959,-178.348,7.365,148.906
C01108=1138.026,183.966,-61.936,-178.350,7.363,148.907
C01109=1138.031,183.697,-61.910,-178.354,7.361,148.907
C01110=1138.036,183.427,-61.885,-178.357,7.358,148.907
C01111=1138.041,183.157,-61.860,-178.360,7.355,148.908
C01112=1138.046,182.887,-61.835,-178.363,7.353,148.908
C01113=1138.051,182.639,-61.812,-178.365,7.351,148.908
C01114=1138.055,182.390,-61.789,-178.369,7.348,148.908
C01115=1138.060,182.141,-61.766,-178.371,7.346,148.909
C01116=1138.064,181.892,-61.742,-178.374,7.344,148.909
C01117=1138.069,181.643,-61.719,-178.377,7.341,148.909
C01118=1138.073,181.394,-61.696,-178.380,7.339,148.909
C01119=1138.078,181.145,-61.673,-178.383,7.336,148.910
C01120=1138.083,180.897,-61.650,-178.385,7.334,148.910
C01121=1138.087,180.648,-61.627,-178.388,7.332,148.910
C01122=1138.092,180.399,-61.604,-178.391,7.330,148.910
C01123=1138.096,180.150,-61.580,-178.394,7.327,148.911
C01124=1138.101,179.900,-61.558,-178.397,7.325,148.911
C01125=1138.105,179.651,-61.535,-178.399,7.323,148.911
C01126=1138.111,179.403,-61.512,-178.402,7.321,148.912
C01127=1138.115,179.154,-61.489,-178.405,7.318,148.912
C01128=1138.119,178.905,-61.466,-178.408,7.315,148.912
C01129=1138.124,178.656,-61.443,-178.411,7.313,148.912
C01130=1138.128,178.407,-61.421,-178.414,7.311,148.912
C01131=1138.134,178.159,-61.398,-178.417,7.309,148.913
C01132=1138.138,177.910,-61.374,-178.419,7.306,148.913
C01133=1138.143,177.660,-61.352,-178.422,7.304,148.913
C01134=1138.147,177.411,-61.329,-178.425,7.302,148.913
C01135=1138.152,177.163,-61.306,-178.428,7.300,148.914
C01136=1138.156,176.914,-61.283,-178.431,7.297,148.914
C01137=1138.161,176.665,-61.261,-178.433,7.295,148.914
C01138=1138.165,176.416,-61.238,-178.436,7.293,148.915
C01139=1138.171,176.168,-61.215,-178.439,7.291,148.915
C01140=1138.175,175.918,-61.193,-178.442,7.288,148.915
C01141=1138.180,175.669,-61.169,-178.445,7.286,148.916
C01142=1138.184,175.420,-61.147,-178.447,7.283,148.916
C01143=1138.189,175.171,-61.124,-178.450,7.282,148.916
C01144=1138.193,174.923,-61.101,-178.453,7.279,148.916
C01145=1138.198,174.673,-61.079,-178.456,7.277,148.917
C01146=1138.202,174.424,-61.056,-178.459,7.275,148.917
C01147=1138.208,174.175,-61.034,-178.461,7.273,148.917
C01148=1138.212,173.927,-61.011,-178.464,7.270,148.917
C01149=1138.217,173.677,-60.988,-178.467,7.268,148.918
C01150=1138.221,173.429,-60.966,-178.470,7.265,148.918
C01151=1138.226,173.180,-60.944,-178.473,7.264,148.918
C01152=1138.230,172.931,-60.921,-178.476,7.261,148.919
C01153=1138.235,172.682,-60.899,-178.478,7.259,148.919
C01154=1138.240,172.433,-60.875,-178.482,7.257,148.919
C01155=1138.244,172.184,-60.853,-178.484,7.255,148.919
C01156=1138.249,171.935,-60.830,-178.487,7.252,148.920
C01157=1138.254,171.686,-60.808,-178.490,7.250,148.920
C01158=1138.258,171.437,-60.786,-178.493,7.248,148.920
C01159=1138.263,171.188,-60.763,-178.495,7.246,148.920
C01160=1138.268,170.939,-60.741,-178.498,7.244,148.921
C01161=1138.272,170.691,-60.719,-178.501,7.241,148.921
C01162=1138.277,170.441,-60.696,-178.504,7.239,148.921
C01163=1138.281,170.193,-60.673,-178.507,7.237,148.922
C01164=1138.287,169.944,-60.651,-178.510,7.235,148.922
C01165=1138.291,169.694,-60.629,-178.512,7.232,148.922
C01166=1138.296,169.446,-60.607,-178.515,7.230,148.923
C01167=1138.301,169.197,-60.584,-178.518,7.228,148.923
C01168=1138.305,168.947,-60.562,-178.521,7.226,148.923
C01169=1138.310,168.699,-60.540,-178.524,7.223,148.923
C01170=1138.314,168.450,-60.518,-178.527,7.222,148.924
C01171=1138.319,168.201,-60.495,-178.529,7.219,148.924
C01172=1138.324,167.952,-60.473,-178.532,7.217,148.924
C01173=1138.328,167.703,-60.452,-178.535,7.215,148.925
C01174=1138.333,167.454,-60.428,-178.538,7.212,148.925
C01175=1138.338,167.205,-60.407,-178.540,7.211,148.925
C01176=1138.342,166.956,-60.385,-178.544,7.208,148.926
C01177=1138.346,166.707,-60.362,-178.546,7.206,148.926
C01178=1138.352,166.458,-60.340,-178.549,7.204,148.926
C01179=1138.356,166.209,-60.317,-178.552,7.202,148.926
C01180=1138.361,165.960,-60.296,-178.554,7.200,148.927
C01181=1138.365,165.711,-60.274,-178.557,7.197,148.927
C01182=1138.370,165.462,-60.252,-178.560,7.195,148.927
C01183=1138.375,165.213,-60.229,-178.563,7.193,148.928
C01184=1138.380,164.964,-60.208,-178.566,7.191,148.928
C01185=1138.384,164.715,-60.186,-178.569,7.188,148.928
C01186=1138.389,164.466,-60.164,-178.572,7.187,148.929
C01187=1138.393,164.217,-60.141,-178.574,7.185,148.929
C01188=1138.398,163.969,-60.120,-178.577,7.182,148.929
C01189=1138.402,163.719,-60.097,-178.580,7.180,148.929
C01190=1138.408,163.470,-60.075,-178.583,7.178,148.930
C01191=1138.412,163.221,-60.053,-178.585,7.176,148.930
C01192=1138.417,162.972,-60.031,-178.588,7.174,148.930
C01193=1138.421,162.723,-60.009,-178.591,7.172,148.931
C01194=1138.426,162.474,-59.988,-178.594,7.170,148.931
C01195=1138.431,162.226,-59.966,-178.597,7.167,148.931
C01196=1138.435,161.976,-59.944,-178.600,7.165,148.932
C01197=1138.440,161.728,-59.922,-178.602,7.163,148.932
C01198=1138.444,161.478,-59.900,-178.605,7.161,148.932
C01199=1138.450,161.229,-59.879,-178.608,7.159,148.932
C01200=1138.454,160.980,-59.857,-178.611,7.156,148.933
C01201=1138.459,160.731,-59.836,-178.614,7.155,148.933
C01202=1138.464,160.483,-59.814,-178.616,7.153,148.933
C01203=1138.468,160.233,-59.792,-178.619,7.150,148.934
C01204=1138.473,159.985,-59.770,-178.622,7.148,148.934
C01205=1138.477,159.735,-59.748,-178.625,7.147,148.934
C01206=1138.482,159.487,-59.726,-178.628,7.144,148.935
C01207=1138.487,159.237,-59.705,-178.630,7.142,148.935
C01208=1138.491,158.988,-59.683,-178.634,7.140,148.935
C01209=1138.496,158.739,-59.662,-178.636,7.138,148.936
C01210=1138.500,158.490,-59.640,-178.639,7.136,148.936
C01211=1138.505,158.241,-59.618,-178.642,7.133,148.936
C01212=1138.510,157.992,-59.597,-178.645,7.131,148.937
C01213=1138.516,157.723,-59.573,-178.648,7.129,148.937
C01214=1138.520,157.454,-59.550,-178.651,7.127,148.937
C01215=1138.526,157.185,-59.527,-178.654,7.125,148.938
C01216=1138.530,156.917,-59.503,-178.657,7.122,148.938
C01217=1138.535,156.667,-59.482,-178.660,7.120,148.938
C01218=1138.540,156.418,-59.460,-178.662,7.118,148.939
C01219=1138.545,156.169,-59.439,-178.666,7.116,148.939
C01220=1138.550,155.920,-59.418,-178.668,7.114,148.939
C01221=1138.554,155.671,-59.396,-178.671,7.112,148.940
C01222=1138.559,155.422,-59.374,-178.674,7.110,148.940
C01223=1138.564,155.173,-59.353,-178.676,7.108,148.940
C01224=1138.568,154.924,-59.332,-178.679,7.106,148.941
C01225=1138.572,154.675,-59.310,-178.682,7.104,148.941
C01226=1138.578,154.426,-59.289,-178.685,7.102,148.941
C01227=1138.583,154.177,-59.267,-178.687,7.100,148.942
C01228=1138.587,153.927,-59.246,-178.691,7.097,148.942
C01229=1138.592,153.679,-59.224,-178.693,7.096,148.942
C01230=1138.596,153.430,-59.204,-178.696,7.094,148.943
C01231=1138.601,153.181,-59.182,-178.699,7.091,148.943
C01232=1138.606,152.931,-59.161,-178.702,7.089,148.943
C01233=1138.611,152.682,-59.139,-178.704,7.088,148.944
C01234=1138.616,152.433,-59.118,-178.708,7.085,148.944
C01235=1138.620,152.185,-59.097,-178.710,7.083,148.944
C01236=1138.625,151.935,-59.076,-178.713,7.082,148.945
C01237=1138.629,151.686,-59.054,-178.716,7.079,148.945
C01238=1138.635,151.437,-59.033,-178.719,7.077,148.945
C01239=1138.639,151.189,-59.012,-178.721,7.075,148.946
C01240=1138.644,150.939,-58.991,-178.724,7.074,148.946
C01241=1138.648,150.690,-58.969,-178.727,7.071,148.946
C01242=1138.653,150.441,-58.948,-178.730,7.070,148.947
C01243=1138.658,150.192,-58.928,-178.732,7.067,148.947
C01244=1138.663,149.943,-58.906,-178.736,7.065,148.947
C01245=1138.668,149.694,-58.885,-178.738,7.063,148.948
C01246=1138.672,149.444,-58.864,-178.741,7.062,148.948
C01247=1138.677,149.196,-58.843,-178.744,7.059,148.948
C01248=1138.682,148.946,-58.822,-178.747,7.057,148.949
C01249=1138.686,148.697,-58.801,-178.749,7.055,148.949
C01250=1138.691,148.449,-58.780,-178.752,7.054,148.949
C01251=1138.696,148.200,-58.759,-178.755,7.051,148.950
C01252=1138.700,147.950,-58.738,-178.758,7.049,148.950
C01253=1138.705,147.701,-58.716,-178.761,7.048,148.951
C01254=1138.709,147.452,-58.696,-178.764,7.045,148.951
C01255=1138.715,147.203,-58.675,-178.766,7.043,148.951
C01256=1138.720,146.954,-58.654,-178.769,7.041,148.951
C01257=1138.724,146.705,-58.633,-178.772,7.040,148.952
C01258=1138.729,146.456,-58.612,-178.775,7.037,148.952
C01259=1138.733,146.207,-58.591,-178.778,7.035,148.953
C01260=1138.738,145.957,-58.570,-178.781,7.034,148.953
C01261=1138.742,145.708,-58.550,-178.783,7.032,148.953
C01262=1138.747,145.460,-58.528,-178.786,7.029,148.954
C01263=1138.753,145.210,-58.507,-178.789,7.027,148.954
C01264=1138.757,144.962,-58.487,-178.791,7.026,148.954
C01265=1138.762,144.712,-58.466,-178.794,7.024,148.955
C01266=1138.767,144.463,-58.445,-178.798,7.021,148.955
C01267=1138.772,144.214,-58.424,-178.800,7.020,148.955
C01268=1138.776,143.965,-58.404,-178.803,7.018,148.956
C01269=1138.781,143.716,-58.383,-178.806,7.016,148.956
C01270=1138.786,143.467,-58.363,-178.809,7.013,148.956
C01271=1138.791,143.218,-58.342,-178.811,7.012,148.957
C01272=1138.795,142.969,-58.321,-178.814,7.010,148.957
C01273=1138.800,142.720,-58.300,-178.817,7.008,148.958
C01274=1138.804,142.470,-58.279,-178.820,7.006,148.958
C01275=1138.809,142.221,-58.259,-178.823,7.004,148.958
C01276=1138.814,141.972,-58.238,-178.825,7.002,148.959
C01277=1138.818,141.723,-58.217,-178.828,7.001,148.959
C01278=1138.823,141.474,-58.196,-178.831,6.998,148.959
C01279=1138.828,141.225,-58.176,-178.834,6.996,148.960
C01280=1138.832,140.976,-58.156,-178.836,6.994,148.960
C01281=1138.838,140.726,-58.135,-178.839,6.993,148.960
C01282=1138.842,140.477,-58.115,-178.842,6.990,148.961
C01283=1138.847,140.228,-58.094,-178.845,6.989,148.961
C01284=1138.852,139.979,-58.074,-178.848,6.987,148.962
C01285=1138.856,139.730,-58.053,-178.851,6.985,148.962
C01286=1138.861,139.481,-58.032,-178.853,6.983,148.962
C01287=1138.866,139.232,-58.012,-178.857,6.981,148.963
C01288=1138.870,138.983,-57.991,-178.859,6.979,148.963
C01289=1138.875,138.734,-57.971,-178.862,6.977,148.963
C01290=1138.881,138.485,-57.951,-178.864,6.975,148.964
C01291=1138.885,138.236,-57.931,-178.867,6.974,148.964
C01292=1138.890,137.987,-57.910,-178.870,6.971,148.964
C01293=1138.895,137.738,-57.890,-178.873,6.970,148.965
C01294=1138.899,137.489,-57.869,-178.876,6.968,148.965
C01295=1138.904,137.239,-57.849,-178.878,6.966,148.966
C01296=1138.909,136.990,-57.829,-178.881,6.964,148.966
C01297=1138.914,136.741,-57.808,-178.884,6.962,148.966
C01298=1138.918,136.492,-57.788,-178.887,6.960,148.967
C01299=1138.923,136.242,-57.768,-178.890,6.959,148.967
C01300=1138.928,135.993,-57.747,-178.893,6.957,148.968
C01301=1138.932,135.744,-57.727,-178.895,6.955,148.968
C01302=1138.937,135.495,-57.706,-178.898,6.952,148.968
C01303=1138.942,135.246,-57.687,-178.901,6.951,148.969
C01304=1138.947,134.997,-57.666,-178.904,6.949,148.969
C01305=1138.952,134.748,-57.646,-178.906,6.947,148.969
C01306=1138.956,134.499,-57.626,-178.909,6.946,148.970
C01307=1138.961,134.250,-57.606,-178.912,6.944,148.970
C01308=1138.965,134.001,-57.585,-178.915,6.941,148.971
C01309=1138.971,133.751,-57.565,-178.918,6.940,148.971
C01310=1138.975,133.502,-57.545,-178.921,6.938,148.971
C01311=1138.981,133.253,-57.525,-178.923,6.936,148.972
C01312=1138.985,133.004,-57.505,-178.926,6.935,148.972
C01313=1138.990,132.755,-57.485,-178.929,6.933,148.972
C01314=1138.994,132.506,-57.465,-178.932,6.930,148.973
C01315=1138.999,132.256,-57.444,-178.935,6.929,148.973
C01316=1139.004,132.007,-57.424,-178.937,6.927,148.974
C01317=1139.009,131.739,-57.403,-178.940,6.925,148.974
C01318=1139.015,131.470,-57.381,-178.944,6.923,148.974
C01319=1139.020,131.202,-57.360,-178.946,6.921,148.975
C01320=1139.025,130.933,-57.339,-178.949,6.919,148.975
C01321=1139.030,130.684,-57.318,-178.952,6.917,148.976
C01322=1139.035,130.434,-57.299,-178.955,6.915,148.976
C01323=1139.039,130.185,-57.278,-178.958,6.913,148.976
C01324=1139.044,129.936,-57.258,-178.960,6.912,148.977
C01325=1139.049,129.688,-57.238,-178.963,6.910,148.977
C01326=1139.054,129.438,-57.219,-178.966,6.908,148.978
C01327=1139.058,129.189,-57.198,-178.969,6.907,148.978
C01328=1139.063,128.939,-57.179,-178.972,6.904,148.978
C01329=1139.068,128.691,-57.160,-178.975,6.902,148.979
C01330=1139.073,128.442,-57.139,-178.977,6.901,148.979
C01331=1139.077,128.192,-57.119,-178.980,6.899,148.980
C01332=1139.082,127.942,-57.100,-178.983,6.897,148.980
C01333=1139.087,127.694,-57.080,-178.986,6.896,148.980
C01334=1139.092,127.445,-57.060,-178.988,6.894,148.981
C01335=1139.097,127.195,-57.041,-178.991,6.892,148.981
C01336=1139.101,126.946,-57.020,-178.994,6.890,148.982
C01337=1139.106,126.697,-57.001,-178.997,6.888,148.982
C01338=1139.111,126.448,-56.981,-179.000,6.886,148.982
C01339=1139.116,126.199,-56.961,-179.002,6.885,148.983
C01340=1139.121,125.950,-56.942,-179.005,6.883,148.983
C01341=1139.126,125.700,-56.922,-179.008,6.881,148.984
C01342=1139.130,125.451,-56.903,-179.011,6.880,148.984
C01343=1139.135,125.203,-56.883,-179.013,6.878,148.984
C01344=1139.140,124.953,-56.863,-179.016,6.876,148.985
C01345=1139.144,124.704,-56.843,-179.019,6.874,148.985
C01346=1139.149,124.454,-56.824,-179.022,6.872,148.986
C01347=1139.154,124.205,-56.805,-179.025,6.870,148.986
C01348=1139.159,123.956,-56.784,-179.028,6.869,148.986
C01349=1139.164,123.707,-56.765,-179.030,6.867,148.987
C01350=1139.168,123.458,-56.746,-179.033,6.865,148.987
C01351=1139.173,123.209,-56.726,-179.036,6.864,148.988
C01352=1139.178,122.960,-56.707,-179.038,6.862,148.988
C01353=1139.183,122.710,-56.687,-179.041,6.860,148.988
C01354=1139.188,122.461,-56.668,-179.044,6.859,148.989
C01355=1139.193,122.212,-56.648,-179.047,6.857,148.989
C01356=1139.197,121.963,-56.628,-179.049,6.855,148.990
C01357=1139.202,121.714,-56.609,-179.053,6.853,148.990
C01358=1139.207,121.465,-56.590,-179.055,6.851,148.990
C01359=1139.212,121.215,-56.570,-179.058,6.849,148.991
C01360=1139.217,120.966,-56.551,-179.061,6.848,148.991
C01361=1139.221,120.717,-56.532,-179.064,6.846,148.992
C01362=1139.226,120.467,-56.512,-179.066,6.844,148.992
C01363=1139.231,120.219,-56.493,-179.069,6.843,148.992
C01364=1139.236,119.969,-56.473,-179.072,6.841,148.993
C01365=1139.240,119.720,-56.454,-179.075,6.839,148.993
C01366=1139.245,119.471,-56.435,-179.077,6.837,148.994
C01367=1139.250,119.221,-56.415,-179.080,6.836,148.994
C01368=1139.255,118.972,-56.396,-179.083,6.834,148.994
C01369=1139.259,118.723,-56.377,-179.085,6.832,148.995
C01370=1139.265,118.474,-56.358,-179.088,6.831,148.995
C01371=1139.270,118.224,-56.338,-179.091,6.829,148.996
C01372=1139.274,117.976,-56.320,-179.094,6.827,148.996
C01373=1139.279,117.726,-56.300,-179.097,6.825,148.996
C01374=1139.284,117.477,-56.281,-179.100,6.824,148.997
C01375=1139.288,117.228,-56.262,-179.103,6.822,148.997
C01376=1139.294,116.979,-56.242,-179.106,6.820,148.998
C01377=1139.298,116.729,-56.223,-179.108,6.818,148.998
C01378=1139.303,116.480,-56.205,-179.111,6.817,148.999
C01379=1139.308,116.231,-56.185,-179.114,6.815,148.999
C01380=1139.313,115.982,-56.166,-179.116,6.813,148.999
C01381=1139.317,115.733,-56.147,-179.119,6.812,149.000
C01382=1139.323,115.484,-56.127,-179.122,6.810,149.000
C01383=1139.327,115.234,-56.109,-179.125,6.808,149.001
C01384=1139.332,114.985,-56.090,-179.127,6.807,149.001
C01385=1139.337,114.735,-56.070,-179.130,6.805,149.001
C01386=1139.342,114.487,-56.051,-179.133,6.803,149.002
C01387=1139.347,114.237,-56.032,-179.136,6.802,149.002
C01388=1139.351,113.988,-56.014,-179.138,6.800,149.003
C01389=1139.356,113.738,-55.994,-179.141,6.798,149.003
C01390=1139.361,113.490,-55.975,-179.144,6.797,149.004
C01391=1139.366,113.240,-55.957,-179.147,6.795,149.004
C01392=1139.371,112.991,-55.937,-179.150,6.794,149.005
C01393=1139.375,112.742,-55.918,-179.152,6.792,149.005
C01394=1139.381,112.492,-55.900,-179.155,6.790,149.005
C01395=1139.385,112.244,-55.881,-179.158,6.789,149.006
C01396=1139.390,111.994,-55.861,-179.161,6.787,149.006
C01397=1139.395,111.745,-55.843,-179.163,6.785,149.007
C01398=1139.400,111.495,-55.824,-179.166,6.783,149.007
C01399=1139.405,111.246,-55.806,-179.169,6.782,149.007
C01400=1139.410,110.997,-55.786,-179.172,6.780,149.008
C01401=1139.414,110.748,-55.767,-179.174,6.778,149.008
C01402=1139.420,110.498,-55.749,-179.177,6.777,149.009
C01403=1139.424,110.249,-55.730,-179.180,6.775,149.009
C01404=1139.429,110.000,-55.711,-179.183,6.774,149.010
C01405=1139.434,109.751,-55.692,-179.186,6.772,149.010
C01406=1139.438,109.501,-55.674,-179.188,6.770,149.010
C01407=1139.444,109.252,-55.655,-179.191,6.769,149.011
C01408=1139.449,109.003,-55.637,-179.194,6.767,149.011
C01409=1139.453,108.754,-55.617,-179.197,6.765,149.012
C01410=1139.458,108.505,-55.599,-179.199,6.764,149.012
C01411=1139.462,108.255,-55.580,-179.202,6.762,149.013
C01412=1139.468,108.006,-55.561,-179.205,6.760,149.013
C01413=1139.472,107.757,-55.543,-179.208,6.759,149.014
C01414=1139.478,107.507,-55.524,-179.211,6.757,149.014
C01415=1139.482,107.258,-55.506,-179.213,6.756,149.014
C01416=1139.487,107.009,-55.487,-179.216,6.754,149.015
C01417=1139.492,106.759,-55.468,-179.219,6.752,149.015
C01418=1139.497,106.511,-55.450,-179.221,6.751,149.016
C01419=1139.502,106.261,-55.432,-179.224,6.750,149.016
C01420=1139.507,106.011,-55.413,-179.227,6.748,149.016
C01421=1139.511,105.744,-55.392,-179.230,6.746,149.017
C01422=1139.517,105.475,-55.372,-179.233,6.744,149.017
C01423=1139.522,105.207,-55.353,-179.236,6.743,149.018
C01424=1139.527,104.938,-55.334,-179.239,6.741,149.018
C01425=1139.532,104.689,-55.314,-179.242,6.740,149.019
C01426=1139.537,104.440,-55.296,-179.244,6.738,149.019
C01427=1139.542,104.191,-55.278,-179.247,6.736,149.020
C01428=1139.547,103.942,-55.259,-179.250,6.735,149.020
C01429=1139.552,103.692,-55.240,-179.253,6.733,149.021
C01430=1139.557,103.443,-55.222,-179.255,6.731,149.021
C01431=1139.561,103.193,-55.204,-179.258,6.730,149.021
C01432=1139.567,102.945,-55.185,-179.261,6.728,149.022
C01433=1139.571,102.695,-55.167,-179.264,6.727,149.022
C01434=1139.576,102.446,-55.149,-179.266,6.726,149.023
C01435=1139.581,102.196,-55.131,-179.269,6.724,149.023
C01436=1139.586,101.947,-55.113,-179.272,6.722,149.024
C01437=1139.591,101.698,-55.093,-179.274,6.721,149.024
C01438=1139.596,101.448,-55.075,-179.277,6.719,149.025
C01439=1139.600,101.199,-55.057,-179.280,6.717,149.025
C01440=1139.605,100.950,-55.039,-179.283,6.716,149.025
C01441=1139.610,100.701,-55.021,-179.286,6.714,149.026
C01442=1139.615,100.451,-55.003,-179.289,6.713,149.026
C01443=1139.620,100.202,-54.984,-179.291,6.711,149.027
C01444=1139.625,99.953,-54.966,-179.294,6.709,149.027
C01445=1139.630,99.704,-54.948,-179.296,6.708,149.028
C01446=1139.635,99.455,-54.930,-179.299,6.707,149.028
C01447=1139.639,99.205,-54.911,-179.302,6.705,149.029
C01448=1139.644,98.956,-54.893,-179.305,6.704,149.029
C01449=1139.649,98.706,-54.875,-179.308,6.702,149.030
C01450=1139.654,98.457,-54.857,-179.310,6.700,149.030
C01451=1139.659,98.208,-54.839,-179.313,6.699,149.030
C01452=1139.664,97.959,-54.821,-179.316,6.697,149.031
C01453=1139.669,97.709,-54.803,-179.319,6.695,149.031
C01454=1139.673,97.460,-54.785,-179.322,6.694,149.032
C01455=1139.678,97.210,-54.767,-179.324,6.693,149.032
C01456=1139.683,96.961,-54.749,-179.327,6.692,149.033
C01457=1139.688,96.712,-54.731,-179.329,6.690,149.033
C01458=1139.693,96.463,-54.713,-179.332,6.688,149.034
C01459=1139.698,96.214,-54.695,-179.335,6.686,149.034
C01460=1139.703,95.964,-54.677,-179.338,6.685,149.035
C01461=1139.707,95.715,-54.658,-179.341,6.684,149.035
C01462=1139.712,95.465,-54.640,-179.344,6.682,149.035
C01463=1139.717,95.216,-54.622,-179.346,6.681,149.036
C01464=1139.722,94.966,-54.605,-179.348,6.679,149.036
C01465=1139.727,94.717,-54.587,-179.351,6.678,149.037
C01466=1139.732,94.468,-54.569,-179.354,6.676,149.037
C01467=1139.737,94.219,-54.551,-179.357,6.675,149.038
C01468=1139.742,93.970,-54.533,-179.360,6.673,149.038
C01469=1139.747,93.721,-54.515,-179.363,6.671,149.039
C01470=1139.752,93.471,-54.497,-179.365,6.670,149.039
C01471=1139.757,93.222,-54.480,-179.368,6.669,149.039
C01472=1139.762,92.972,-54.462,-179.371,6.667,149.040
C01473=1139.767,92.723,-54.444,-179.373,6.666,149.041
C01474=1139.772,92.474,-54.426,-179.376,6.664,149.041
C01475=1139.776,92.224,-54.408,-179.379,6.662,149.041
C01476=1139.781,91.974,-54.390,-179.382,6.661,149.042
C01477=1139.785,91.726,-54.373,-179.384,6.660,149.042
C01478=1139.790,91.476,-54.355,-179.387,6.659,149.043
C01479=1139.795,91.227,-54.337,-179.390,6.657,149.043
C01480=1139.800,90.977,-54.320,-179.393,6.655,149.044
C01481=1139.805,90.728,-54.302,-179.395,6.654,149.044
C01482=1139.810,90.479,-54.284,-179.398,6.652,149.045
C01483=1139.816,90.229,-54.267,-179.401,6.651,149.045
C01484=1139.820,89.980,-54.249,-179.403,6.650,149.046
C01485=1139.825,89.731,-54.231,-179.406,6.648,149.046
C01486=1139.830,89.481,-54.214,-179.409,6.646,149.046
C01487=1139.835,89.232,-54.196,-179.412,6.645,149.047
C01488=1139.840,88.983,-54.178,-179.415,6.643,149.048
C01489=1139.845,88.733,-54.161,-179.417,6.643,149.048
C01490=1139.850,88.484,-54.143,-179.420,6.641,149.048
C01491=1139.854,88.235,-54.125,-179.422,6.639,149.049
C01492=1139.859,87.985,-54.108,-179.425,6.638,149.049
C01493=1139.865,87.737,-54.090,-179.428,6.636,149.050
C01494=1139.870,87.487,-54.073,-179.431,6.635,149.050
C01495=1139.874,87.238,-54.056,-179.433,6.634,149.051
C01496=1139.879,86.989,-54.039,-179.436,6.632,149.051
C01497=1139.884,86.739,-54.021,-179.439,6.630,149.052
C01498=1139.889,86.490,-54.003,-179.442,6.629,149.052
C01499=1139.894,86.241,-53.986,-179.445,6.628,149.053
C01500=1139.898,85.992,-53.968,-179.447,6.627,149.053
C01501=1139.904,85.742,-53.951,-179.450,6.625,149.053
C01502=1139.909,85.493,-53.933,-179.452,6.623,149.054
C01503=1139.913,85.243,-53.916,-179.456,6.622,149.055
C01504=1139.918,84.993,-53.899,-179.458,6.621,149.055
C01505=1139.923,84.744,-53.881,-179.460,6.619,149.055
C01506=1139.928,84.495,-53.864,-179.463,6.618,149.056
C01507=1139.933,84.246,-53.847,-179.466,6.617,149.056
C01508=1139.938,83.996,-53.829,-179.469,6.615,149.057
C01509=1139.943,83.747,-53.811,-179.471,6.614,149.057
C01510=1139.948,83.498,-53.795,-179.474,6.612,149.058
C01511=1139.953,83.248,-53.777,-179.477,6.611,149.058
C01512=1139.957,82.999,-53.760,-179.480,6.609,149.059
C01513=1139.962,82.749,-53.743,-179.483,6.608,149.059
C01514=1139.968,82.501,-53.725,-179.485,6.607,149.060
C01515=1139.972,82.251,-53.708,-179.488,6.605,149.060
C01516=1139.978,82.001,-53.691,-179.491,6.604,149.061
C01517=1139.983,81.752,-53.673,-179.494,6.602,149.061
C01518=1139.987,81.503,-53.656,-179.496,6.601,149.062
C01519=1139.992,81.253,-53.639,-179.499,6.600,149.062
C01520=1139.996,81.004,-53.622,-179.501,6.598,149.062
C01521=1140.002,80.755,-53.605,-179.504,6.597,149.063
C01522=1140.007,80.505,-53.588,-179.507,6.596,149.064
C01523=1140.012,80.256,-53.571,-179.509,6.594,149.064
C01524=1140.017,80.007,-53.553,-179.512,6.593,149.064
C01525=1140.022,79.739,-53.535,-179.515,6.591,149.065
C01526=1140.028,79.470,-53.517,-179.518,6.590,149.065
C01527=1140.033,79.201,-53.498,-179.521,6.588,149.066
C01528=1140.038,78.933,-53.480,-179.524,6.587,149.067
C01529=1140.043,78.683,-53.463,-179.527,6.585,149.067
C01530=1140.048,78.434,-53.446,-179.529,6.585,149.068
C01531=1140.053,78.185,-53.428,-179.532,6.583,149.068
C01532=1140.058,77.936,-53.412,-179.535,6.581,149.068
C01533=1140.063,77.686,-53.395,-179.538,6.580,149.069
C01534=1140.068,77.437,-53.378,-179.540,6.579,149.069
C01535=1140.073,77.187,-53.361,-179.543,6.577,149.070
C01536=1140.078,76.938,-53.344,-179.546,6.576,149.070
C01537=1140.083,76.689,-53.326,-179.548,6.575,149.071
C01538=1140.087,76.439,-53.310,-179.551,6.573,149.071
C01539=1140.092,76.190,-53.293,-179.554,6.572,149.072
C01540=1140.098,75.941,-53.276,-179.557,6.570,149.072
C01541=1140.103,75.691,-53.259,-179.559,6.569,149.073
C01542=1140.107,75.442,-53.242,-179.562,6.568,149.073
C01543=1140.112,75.193,-53.226,-179.565,6.566,149.074
C01544=1140.118,74.943,-53.209,-179.568,6.565,149.074
C01545=1140.122,74.693,-53.192,-179.570,6.564,149.075
C01546=1140.127,74.444,-53.175,-179.572,6.562,149.075
C01547=1140.132,74.195,-53.159,-179.576,6.561,149.076
C01548=1140.137,73.945,-53.142,-179.578,6.560,149.076
C01549=1140.142,73.696,-53.125,-179.581,6.559,149.077
C01550=1140.147,73.447,-53.108,-179.584,6.557,149.077
C01551=1140.152,73.197,-53.091,-179.586,6.556,149.078
C01552=1140.157,72.948,-53.074,-179.589,6.555,149.078
C01553=1140.162,72.699,-53.058,-179.591,6.553,149.079
C01554=1140.167,72.449,-53.041,-179.595,6.552,149.079
C01555=1140.172,72.199,-53.024,-179.597,6.551,149.080
C01556=1140.177,71.951,-53.008,-179.600,6.549,149.080
C01557=1140.182,71.701,-52.991,-179.602,6.548,149.081
C01558=1140.186,71.451,-52.974,-179.605,6.547,149.081
C01559=1140.191,71.203,-52.958,-179.608,6.545,149.082
C01560=1140.197,70.953,-52.940,-179.610,6.544,149.082
C01561=1140.201,70.703,-52.924,-179.613,6.543,149.083
C01562=1140.206,70.454,-52.908,-179.616,6.542,149.083
C01563=1140.211,70.204,-52.891,-179.619,6.540,149.084
C01564=1140.216,69.955,-52.874,-179.621,6.539,149.084
C01565=1140.221,69.706,-52.858,-179.624,6.538,149.085
C01566=1140.226,69.456,-52.841,-179.627,6.536,149.085
C01567=1140.232,69.207,-52.824,-179.629,6.535,149.086
C01568=1140.236,68.957,-52.808,-179.632,6.534,149.086
C01569=1140.241,68.708,-52.792,-179.635,6.532,149.087
C01570=1140.246,68.459,-52.775,-179.638,6.531,149.087
C01571=1140.250,68.209,-52.759,-179.640,6.530,149.088
C01572=1140.257,67.960,-52.742,-179.642,6.528,149.088
C01573=1140.261,67.710,-52.726,-179.646,6.527,149.089
C01574=1140.265,67.461,-52.709,-179.648,6.526,149.089
C01575=1140.271,67.212,-52.693,-179.651,6.525,149.090
C01576=1140.275,66.962,-52.677,-179.654,6.523,149.090
C01577=1140.281,66.713,-52.660,-179.656,6.522,149.091
C01578=1140.286,66.463,-52.643,-179.659,6.521,149.091
C01579=1140.291,66.215,-52.627,-179.661,6.520,149.092
C01580=1140.296,65.964,-52.611,-179.664,6.519,149.092
C01581=1140.301,65.716,-52.595,-179.667,6.517,149.093
C01582=1140.305,65.466,-52.578,-179.669,6.516,149.093
C01583=1140.311,65.216,-52.562,-179.672,6.515,149.094
C01584=1140.316,64.967,-52.545,-179.675,6.513,149.094
C01585=1140.320,64.717,-52.529,-179.677,6.512,149.095
C01586=1140.326,64.468,-52.513,-179.680,6.511,149.095
C01587=1140.330,64.219,-52.496,-179.683,6.509,149.096
C01588=1140.335,63.969,-52.481,-179.685,6.509,149.096
C01589=1140.340,63.720,-52.464,-179.688,6.507,149.097
C01590=1140.345,63.471,-52.448,-179.691,6.506,149.097
C01591=1140.350,63.221,-52.432,-179.693,6.505,149.098
C01592=1140.356,62.972,-52.415,-179.696,6.503,149.098
C01593=1140.360,62.722,-52.399,-179.699,6.503,149.099
C01594=1140.365,62.473,-52.383,-179.702,6.501,149.099
C01595=1140.370,62.223,-52.367,-179.704,6.499,149.100
C01596=1140.375,61.974,-52.350,-179.706,6.499,149.100
C01597=1140.380,61.724,-52.334,-179.710,6.497,149.101
C01598=1140.385,61.475,-52.318,-179.712,6.496,149.101
C01599=1140.390,61.225,-52.302,-179.715,6.495,149.102
C01600=1140.395,60.976,-52.286,-179.718,6.493,149.102
C01601=1140.400,60.727,-52.270,-179.720,6.493,149.103
C01602=1140.405,60.477,-52.254,-179.723,6.491,149.103
C01603=1140.410,60.228,-52.238,-179.726,6.490,149.104
C01604=1140.415,59.978,-52.221,-179.728,6.489,149.104
C01605=1140.420,59.729,-52.206,-179.731,6.487,149.105
C01606=1140.425,59.480,-52.189,-179.733,6.486,149.105
C01607=1140.430,59.230,-52.173,-179.736,6.485,149.106
C01608=1140.435,58.981,-52.157,-179.739,6.483,149.106
C01609=1140.440,58.731,-52.141,-179.741,6.483,149.107
C01610=1140.445,58.482,-52.126,-179.744,6.481,149.107
C01611=1140.450,58.232,-52.109,-179.747,6.480,149.108
C01612=1140.455,57.983,-52.093,-179.749,6.479,149.108
C01613=1140.461,57.734,-52.078,-179.753,6.478,149.109
C01614=1140.465,57.484,-52.061,-179.755,6.477,149.109
C01615=1140.470,57.235,-52.046,-179.757,6.475,149.110
C01616=1140.475,56.985,-52.030,-179.760,6.475,149.110
C01617=1140.480,56.736,-52.014,-179.763,6.473,149.111
C01618=1140.485,56.487,-51.998,-179.766,6.471,149.111
C01619=1140.490,56.237,-51.982,-179.768,6.471,149.112
C01620=1140.495,55.988,-51.966,-179.771,6.469,149.112
C01621=1140.500,55.738,-51.950,-179.773,6.468,149.113
C01622=1140.505,55.488,-51.934,-179.776,6.467,149.113
C01623=1140.510,55.239,-51.919,-179.779,6.466,149.114
C01624=1140.515,54.989,-51.902,-179.781,6.465,149.114
C01625=1140.520,54.740,-51.887,-179.784,6.463,149.115
C01626=1140.525,54.491,-51.872,-179.787,6.462,149.116
C01627=1140.530,54.241,-51.856,-179.789,6.461,149.116
C01628=1140.535,53.992,-51.839,-179.792,6.460,149.116
C01629=1140.540,53.724,-51.822,-179.795,6.459,149.117
C01630=1140.546,53.454,-51.806,-179.798,6.457,149.117
C01631=1140.552,53.186,-51.789,-179.801,6.456,149.118
C01632=1140.557,52.917,-51.772,-179.803,6.455,149.119
C01633=1140.561,52.668,-51.757,-179.806,6.454,149.119
C01634=1140.567,52.418,-51.741,-179.808,6.453,149.120
C01635=1140.572,52.169,-51.725,-179.811,6.451,149.120
C01636=1140.577,51.919,-51.709,-179.814,6.450,149.121
C01637=1140.582,51.670,-51.693,-179.817,6.449,149.121
C01638=1140.587,51.421,-51.678,-179.819,6.447,149.122
C01639=1140.591,51.171,-51.662,-179.822,6.447,149.122
C01640=1140.597,50.921,-51.647,-179.825,6.445,149.123
C01641=1140.602,50.672,-51.631,-179.827,6.445,149.123
C01642=1140.607,50.423,-51.616,-179.830,6.443,149.124
C01643=1140.612,50.173,-51.600,-179.832,6.442,149.124
C01644=1140.617,49.923,-51.585,-179.835,6.441,149.125
C01645=1140.622,49.675,-51.568,-179.838,6.440,149.125
C01646=1140.627,49.426,-51.553,-179.840,6.439,149.126
C01647=1140.632,49.175,-51.537,-179.843,6.438,149.126
C01648=1140.637,48.926,-51.522,-179.846,6.437,149.127
C01649=1140.642,48.677,-51.507,-179.848,6.436,149.127
C01650=1140.647,48.428,-51.491,-179.851,6.434,149.128
C01651=1140.652,48.177,-51.475,-179.854,6.433,149.129
C01652=1140.656,47.928,-51.460,-179.856,6.432,149.129
C01653=1140.662,47.679,-51.445,-179.859,6.430,149.129
C01654=1140.667,47.429,-51.430,-179.862,6.430,149.130
C01655=1140.671,47.179,-51.414,-179.864,6.428,149.131
C01656=1140.677,46.930,-51.399,-179.866,6.427,149.131
C01657=1140.682,46.680,-51.383,-179.870,6.426,149.132
C01658=1140.687,46.431,-51.368,-179.872,6.425,149.132
C01659=1140.692,46.182,-51.353,-179.875,6.424,149.133
C01660=1140.697,45.933,-51.338,-179.877,6.423,149.133
C01661=1140.702,45.683,-51.322,-179.880,6.422,149.134
C01662=1140.707,45.433,-51.306,-179.882,6.421,149.134
C01663=1140.712,45.184,-51.291,-179.885,6.419,149.135
C01664=1140.717,44.935,-51.276,-179.888,6.419,149.135
C01665=1140.722,44.685,-51.261,-179.890,6.417,149.136
C01666=1140.727,44.435,-51.245,-179.893,6.417,149.136
C01667=1140.732,44.185,-51.230,-179.896,6.415,149.137
C01668=1140.737,43.936,-51.215,-179.898,6.414,149.138
C01669=1140.742,43.687,-51.199,-179.901,6.413,149.138
C01670=1140.747,43.437,-51.185,-179.903,6.412,149.138
C01671=1140.753,43.188,-51.169,-179.907,6.411,149.139
C01672=1140.757,42.939,-51.154,-179.909,6.410,149.140
C01673=1140.762,42.689,-51.138,-179.911,6.408,149.140
C01674=1140.767,42.440,-51.123,-179.914,6.408,149.141
C01675=1140.772,42.190,-51.108,-179.917,6.406,149.141
C01676=1140.777,41.940,-51.093,-179.919,6.405,149.142
C01677=1140.782,41.691,-51.078,-179.922,6.404,149.142
C01678=1140.787,41.442,-51.063,-179.924,6.403,149.143
C01679=1140.793,41.192,-51.048,-179.927,6.402,149.143
C01680=1140.797,40.943,-51.033,-179.930,6.401,149.144
C01681=1140.803,40.693,-51.017,-179.932,6.400,149.144
C01682=1140.808,40.444,-51.003,-179.935,6.399,149.145
C01683=1140.813,40.194,-50.987,-179.937,6.398,149.145
C01684=1140.817,39.945,-50.972,-179.940,6.397,149.146
C01685=1140.823,39.695,-50.957,-179.943,6.396,149.146
C01686=1140.828,39.445,-50.942,-179.946,6.395,149.147
C01687=1140.833,39.196,-50.927,-179.948,6.394,149.147
C01688=1140.838,38.946,-50.912,-179.951,6.392,149.148
C01689=1140.843,38.697,-50.897,-179.953,6.392,149.149
C01690=1140.848,38.448,-50.882,-179.956,6.390,149.149
C01691=1140.853,38.198,-50.868,-179.959,6.389,149.150
C01692=1140.858,37.949,-50.852,-179.961,6.389,149.150
C01693=1140.863,37.699,-50.838,-179.963,6.387,149.151
C01694=1140.869,37.450,-50.822,-179.966,6.387,149.151
C01695=1140.874,37.200,-50.808,-179.969,6.385,149.152
C01696=1140.878,36.951,-50.793,-179.971,6.384,149.152
C01697=1140.884,36.701,-50.777,-179.974,6.383,149.153
C01698=1140.889,36.452,-50.763,-179.976,6.382,149.153
C01699=1140.894,36.202,-50.747,-179.980,6.381,149.154
C01700=1140.899,35.953,-50.733,-179.982,6.380,149.154
C01701=1140.904,35.704,-50.718,-179.984,6.379,149.155
C01702=1140.909,35.453,-50.703,-179.987,6.378,149.155
C01703=1140.914,35.204,-50.688,-179.989,6.377,149.156
C01704=1140.919,34.955,-50.674,-179.992,6.375,149.156
C01705=1140.924,34.705,-50.658,-179.995,6.375,149.157
C01706=1140.929,34.456,-50.644,-179.998,6.373,149.158
C01707=1140.934,34.206,-50.630,-180.000,6.372,149.158
C01708=1140.940,33.956,-50.614,179.998,6.372,149.159
C01709=1140.945,33.707,-50.600,179.995,6.370,149.159
C01710=1140.949,33.458,-50.585,179.992,6.370,149.160
C01711=1140.954,33.208,-50.571,179.989,6.368,149.160
C01712=1140.960,32.959,-50.555,179.987,6.367,149.161
C01713=1140.964,32.709,-50.541,179.984,6.366,149.161
C01714=1140.969,32.459,-50.527,179.982,6.365,149.162
C01715=1140.974,32.210,-50.512,179.980,6.365,149.162
C01716=1140.980,31.960,-50.497,179.976,6.363,149.163
C01717=1140.985,31.710,-50.482,179.974,6.363,149.163
C01718=1140.989,31.461,-50.467,179.971,6.361,149.164
C01719=1140.994,31.211,-50.453,179.969,6.360,149.165
C01720=1141.000,30.963,-50.438,179.967,6.360,149.165
C01721=1141.005,30.713,-50.424,179.963,6.358,149.166
C01722=1141.010,30.463,-50.409,179.961,6.358,149.166
C01723=1141.015,30.214,-50.395,179.959,6.356,149.167
C01724=1141.020,29.965,-50.380,179.956,6.355,149.167
C01725=1141.026,29.715,-50.365,179.954,6.355,149.168
C01726=1141.030,29.465,-50.351,179.950,6.353,149.168
C01727=1141.035,29.216,-50.336,179.948,6.353,149.169
C01728=1141.040,28.966,-50.322,179.946,6.351,149.169
C01729=1141.045,28.716,-50.307,179.943,6.350,149.170
C01730=1141.051,28.467,-50.293,179.941,6.350,149.170
C01731=1141.056,28.218,-50.278,179.938,6.348,149.171
C01732=1141.061,27.968,-50.264,179.935,6.348,149.172
C01733=1141.066,27.699,-50.249,179.933,6.346,149.172
C01734=1141.071,27.430,-50.233,179.930,6.346,149.173
C01735=1141.077,27.161,-50.217,179.927,6.344,149.173
C01736=1141.083,26.891,-50.202,179.925,6.343,149.174
C01737=1141.087,26.642,-50.187,179.922,6.342,149.174
C01738=1141.093,26.393,-50.173,179.919,6.341,149.175
C01739=1141.098,26.144,-50.159,179.917,6.341,149.175
C01740=1141.103,25.894,-50.144,179.914,6.339,149.176
C01741=1141.108,25.644,-50.130,179.912,6.338,149.177
C01742=1141.113,25.395,-50.116,179.909,6.337,149.177
C01743=1141.118,25.145,-50.101,179.906,6.336,149.178
C01744=1141.124,24.896,-50.086,179.904,6.336,149.178
C01745=1141.129,24.646,-50.072,179.901,6.334,149.179
C01746=1141.134,24.397,-50.058,179.899,6.334,149.179
C01747=1141.139,24.147,-50.043,179.896,6.333,149.180
C01748=1141.144,23.897,-50.029,179.893,6.331,149.180
C01749=1141.149,23.648,-50.015,179.891,6.331,149.181
C01750=1141.154,23.399,-50.001,179.889,6.330,149.181
C01751=1141.159,23.149,-49.987,179.886,6.329,149.182
C01752=1141.164,22.899,-49.972,179.883,6.328,149.182
C01753=1141.169,22.649,-49.958,179.881,6.327,149.183
C01754=1141.175,22.400,-49.944,179.878,6.326,149.184
C01755=1141.179,22.151,-49.930,179.876,6.325,149.184
C01756=1141.184,21.901,-49.916,179.873,6.324,149.185
C01757=1141.189,21.651,-49.901,179.870,6.323,149.185
C01758=1141.195,21.402,-49.887,179.868,6.322,149.186
C01759=1141.200,21.153,-49.873,179.866,6.322,149.186
C01760=1141.205,20.903,-49.859,179.863,6.320,149.187
C01761=1141.210,20.653,-49.845,179.860,6.319,149.187
C01762=1141.215,20.404,-49.831,179.858,6.319,149.188
C01763=1141.220,20.154,-49.816,179.855,6.317,149.188
C01764=1141.225,19.905,-49.803,179.853,6.317,149.189
C01765=1141.229,19.655,-49.788,179.850,6.316,149.189
C01766=1141.235,19.406,-49.775,179.847,6.315,149.190
C01767=1141.240,19.157,-49.760,179.845,6.314,149.191
C01768=1141.245,18.906,-49.747,179.843,6.313,149.191
C01769=1141.251,18.657,-49.733,179.839,6.312,149.192
C01770=1141.256,18.408,-49.718,179.837,6.311,149.192
C01771=1141.261,18.158,-49.704,179.835,6.310,149.193
C01772=1141.266,17.908,-49.690,179.832,6.309,149.193
C01773=1141.271,17.659,-49.676,179.830,6.308,149.194
C01774=1141.276,17.409,-49.662,179.827,6.308,149.195
C01775=1141.281,17.159,-49.649,179.824,6.306,149.195
C01776=1141.286,16.910,-49.635,179.822,6.305,149.195
C01777=1141.291,16.661,-49.621,179.819,6.305,149.196
C01778=1141.296,16.411,-49.606,179.817,6.303,149.197
C01779=1141.302,16.162,-49.592,179.814,6.303,149.197
C01780=1141.307,15.912,-49.579,179.812,6.302,149.198
C01781=1141.312,15.662,-49.565,179.810,6.301,149.198
C01782=1141.317,15.413,-49.551,179.806,6.300,149.199
C01783=1141.322,15.164,-49.537,179.804,6.299,149.199
C01784=1141.327,14.913,-49.523,179.802,6.298,149.200
C01785=1141.333,14.664,-49.509,179.799,6.297,149.200
C01786=1141.337,14.414,-49.495,179.797,6.296,149.201
C01787=1141.342,14.165,-49.482,179.794,6.296,149.202
C01788=1141.348,13.915,-49.468,179.792,6.295,149.202
C01789=1141.353,13.666,-49.454,179.789,6.294,149.203
C01790=1141.358,13.417,-49.440,179.786,6.293,149.203
C01791=1141.363,13.167,-49.427,179.784,6.292,149.204
C01792=1141.368,12.917,-49.413,179.781,6.291,149.204
C01793=1141.373,12.668,-49.399,179.779,6.290,149.205
C01794=1141.378,12.418,-49.385,179.777,6.289,149.205
C01795=1141.384,12.169,-49.372,179.774,6.289,149.206
C01796=1141.388,11.919,-49.358,179.771,6.287,149.206
C01797=1141.393,11.669,-49.344,179.769,6.287,149.207
C01798=1141.399,11.420,-49.330,179.766,6.286,149.208
C01799=1141.403,11.171,-49.317,179.764,6.285,149.208
C01800=1141.409,10.921,-49.303,179.761,6.284,149.209
C01801=1141.414,10.671,-49.289,179.759,6.283,149.209
C01802=1141.419,10.421,-49.276,179.756,6.282,149.210
C01803=1141.424,10.172,-49.262,179.753,6.281,149.210
C01804=1141.429,9.922,-49.248,179.751,6.280,149.211
C01805=1141.435,9.673,-49.235,179.749,6.280,149.211
